# B&R Automation Studio project PT_KB_V01 (part 8)

### PGRad_Process.typ - not listed in the package file held
```iecst
TYPE
	E_RegulacijaBRB2 :
		( (* Regulaciona petlja pumpe koja doprema vodu iz BRB2. *) (* -------------------------------------------------------------------------- *) (* 1) Glavna stanja, izbor izvora i izbor aktivne opreme                     *)
		BRB2_00_NEAKTIVNA,
		BRB2_01_REG_PROTOK, (* Protok ka Podstanici/Hotelu. *)
		BRB2_02_REG_NIVO, (* Nivo prihvatnog suda. *)
		BRB2_03_REG_TEMPERATURA (* Temperatura sekundara izmenjivaca. *)
		);
	E_PGRad_State :
		( (* Glavna procesna stanja rada Podstanice prema izabranom izvoru. *)
		PG_00_Stand_By, (* Bez aktivnog izvora; izlazi su u bezbednom stanju i ceka se izbor/start. *)
		PG_01_Priprema_BRB2, (* Pokrece BRB2 i priprema ulaznu granu do potvrde pritiska/protoka. *)
		PG_02_Rad_BRB2, (* BRB2 napaja tank; aktivni su regulacija ulaza, izlazna pumpa i odzracivanje. *)
		PG_03_Zaustavljanje_BRB2, (* Kontrolisano ukida zahtev BRB2 i zatvara pripadajuce ventile. *)
		PG_11_Priprema_IEBKB1, (* Priprema IEBKB1 granu pre dozvole punjenja prihvatnog tanka. *)
		PG_12_Rad_IEBKB1, (* IEBKB1 je aktivni izvor i Podstanica vodi lokalnu regulaciju. *)
		PG_13_Zaustavljanje_IEBKB1, (* Kontrolisano zaustavlja IEBKB1 i zatvara njegovu ulaznu granu. *)
		PG_14_Transfer_IEBKB1_BRB2 (* Prebacuje napajanje sa IEBKB1 na prethodno pripremljeni BRB2. *)
		);
	E_BRB2PreparationState :
		( (* Stanja paralelne pripreme BRB2 pre transfera izvora. *)
		BRB2_PREP_00_IDLE, (* Priprema nije trazena; resetuju se privremene potvrde. *)
		BRB2_PREP_10_START, (* Poslat je start zahtev i ceka se potvrda protoka BRB2. *)
		BRB2_PREP_20_ZAGREVANJE, (* BRB2 ispira/zagreva cev do minimalne temperature. *)
		BRB2_PREP_30_SPReady, (* Protok i temperatura su potvrdeni; transfer izvora je dozvoljen. *)
		BRB2_PREP_40_STOPPING, (* Priprema se kontrolisano prekida i ceka se potvrda stopa. *)
		BRB2_PREP_90_FAULT (* Priprema je blokirana timeout-om ili procesnim interlockom. *)
		);
	E_RegulacionaVarijanta :
		( (* Izbor procesne velicine koju Podstanica regulise. *)
		_00_neaktivan, (* 0 - sve ugaseno, ni jedna varijanta nije izabrana. *)
		_01_REG_PRITISAK, (* 1 - PT vodi, prati zadati pritisak. *)
		_02_REG_NIVO (* 2 - PT vodi nivo prihvatnog tanka preko izlazne pumpe. *)
		);
	E_SelektovaniIzvor :
		( (* Izbor aktivnog izvora termalne vode za Podstanicu. *)
		_00_IZVOR_NIJE_IZABRAN, (* 0 - rezervisano za inicijalizaciju i dijagnostiku; binarni HMI selektor ne zadaje ovu vrednost. *)
		_01_BRB2, (* 1 - BRB2 kao izvor. *)
		_02_IEBKB1 (* 2 - IEBKB1 kao izvor. *)
		);
	E_AktivnaPumpaIzlazTanka :
		( (* Izbor aktivne izlazne pumpe prihvatnog tanka. *)
		_00_nijedna, (* 0 - nijedna pumpa aktivna na izlazu iz tanka. *)
		_01_Pu_PG_01, (* 1 - Pu_PG_01 aktivna. *)
		_02_Pu_PG_02 (* 2 - Pu_PG_02 aktivna. *)
		);
	E_AktivniPropVentilUlazTanka :
		( (* Izbor aktivnog proporcionalnog ventila na ulazu u tank. *) (* -------------------------------------------------------------------------- *) (* 2) Retentivni parametri procesa i pomocne runtime strukture                *)
		_00_PROP_VENTIL_NIJE_IZABRAN, (* 0 - nijedan prop. ventil nije izabran. *)
		_01_PG_PV01, (* 1 - PG_PV01 aktivan. *)
		_02_PG_PV02 (* 2 - PG_PV02 aktivan. *)
		);
	typCmdRetainUlazniVentiliPGRad : 	STRUCT  (* Zapamceni zahtevi bistabilnih ulaznih ventila PG_V01 i PG_V02. *)
		V01_Open : BOOL; (* PG_V01 - zapamceni zahtev IEBKB1 ulaznog ventila. *)
		V02_Open : BOOL; (* PG_V02 - zapamceni zahtev BRB2 ulaznog ventila. *)
	END_STRUCT;
	typParAirReleaseModePGRad : 	STRUCT  (* Parametri odzracivanja za jedan izvor vode. *)
		PV03 : typParAirRelease; (* Odzracivanje na ulazu termalne vode u podstanicu. *)
		PV04 : typParAirRelease; (* Odzracivanje na ulazu termalne vode u prihvatni tank. *)
	END_STRUCT;
	typParAirReleasePGRad : 	STRUCT  (* Grupisani parametri odzracivanja prema aktivnom izvoru. *)
		BRB2 : typParAirReleaseModePGRad; (* Parametri rada sa izvorom BRB2. *)
		IEBKB1 : typParAirReleaseModePGRad; (* Parametri rada sa izvorom IEBKB1. *)
	END_STRUCT;
	typTimeSPPGRad : 	STRUCT  (* Grupisani vremenski SP parametri u sekundama. *)
		PrelazPV05Cuvar_s : REAL; (* Vreme PT06 SP rampe [s]. *)
		OverlapPumpi_s : REAL; (* Maksimalno vreme paralelnog rada pri rotaciji [s]. *)
		AutoRestartDelay_s : REAL; (* Zadrzavanje pre automatskog starta [s]. *)
		ValvePositionTimeout_s : REAL; (* Maksimalno vreme hoda ventila [s]. *)
		InterlockDebounce_s : REAL; (* Vreme potvrde interlock povratnog signala [s]. *)
	END_STRUCT;
	typParBRB2PreparationPGRad : 	STRUCT  (* Paralelna priprema BRB2 dok IEBKB1 snabdeva tank. *)
		MinTemperature_degC : REAL; (* Minimalna temperatura TT_PG_07 za spremnost BRB2. *)
		MinFlow_lps : REAL; (* Minimalni potvrdeni protok BRB2 tokom zagrevanja. *)
		FlowTimeout_s : REAL; (* Maksimalno cekanje potvrde protoka nakon starta BRB2. *)
		TemperatureAlarm_s : REAL; (* Vreme do alarma ako temperatura nije dostignuta. *)
		TemperatureStopDelay_s : REAL; (* Dodatno vreme od alarma do kontrolisanog stopa. *)
		PressureAlarmDelay_s : REAL; (* Vreme visokog PT06 do alarma. *)
		PressureStopDelay_s : REAL; (* Dodatno vreme visokog PT06 do kontrolisanog stopa. *)
	END_STRUCT;
	typParTransferPGRad : 	STRUCT  (* Parametri transfera IEBKB1 na pripremljeni BRB2. *)
		PV05StartPressure_bar : REAL; (* Pocetni PT06 SP regulatora PG_PV05. *)
		PV05FinalPressure_bar : REAL; (* Krajnji PT06 SP regulatora PG_PV05. *)
		TankInletPressure_bar : REAL; (* Stalni PT04 SP aktivnog PG_PV01/PV02. *)
		PressureRamp_s : REAL; (* Trajanje rampe PT06 SP-a. *)
		FlowTimeout_s : REAL; (* Maksimalno cekanje potvrde BRB2 protoka pri transferu. *)
		PV05ClosedPercent : REAL; (* Otvorenost ispod koje se drenaÅ¾a smatra zatvorenom. *)
	END_STRUCT;
	typParPGRad : 	STRUCT  (* Zbirni procesni, vremenski i odzracni parametri Podstanice. *)
		SetPritisakPotisa : REAL; (* Zadati pritisak potisa glavne pumpe [bar]. *)
		MinProtok : REAL; (* Donja granica protoka. *)
		MaxProtok : REAL; (* Gornja granica protoka. *)
		MinFR_Pumpe : REAL; (* Minimalna frekvencija PID izlaza pumpi [Hz]. *)
		MaxFR_Pumpe : REAL; (* Maksimalna frekvencija PID izlaza pumpi [Hz]. *)
		SetPointNivoTanka : REAL; (* Ciljani nivo prihvatnog tanka [m]. *)
		SetPointNivoTankaUpozorenje : REAL; (* Informativni prag blizine fizickog preliva (~2.15-2.2m stvarnog preliva) [m]. *)
		SetPointMinTempIspiranja : REAL; (* Minimalna temperatura za zavrsetak ispiranja [degC]. *)
		SetPointPritisakPV05Ispiranje : REAL; (* PT06 SP tokom preispiranja [bar]. *)
		SetPointPritisakUlazTanka : REAL; (* PT04 SP aktivnog ulaznog ventila [bar]. *)
		SetPointMaxPritisakDolaznaCev : REAL; (* PT06 SP cuvara instalacije [bar]. *)
		PocetnaFrekvencaIzlaznePumpe : REAL; (* PID tracking frekvenca pri startu [Hz]. *)
		MaxOtvorPropZaZatvaranje : REAL; (* Najveca otvorenost za potvrdu zatvaranja [%]. *)
		BRB2Preparation : typParBRB2PreparationPGRad; (* Parametri nezavisnog zagrevanja BRB2. *)
		Transfer : typParTransferPGRad; (* Parametri kontrolisanog transfera izvora. *)
		TimeSP : typTimeSPPGRad; (* RETAIN vremenski SP parametri u sekundama. *)
		AirRelease : typParAirReleasePGRad; (* RETAIN parametri PV03/PV04 za oba izvora. *)
	END_STRUCT;
	typCtrlAirReleasePGRad : 	STRUCT  (* HMI i servisne komande jednog odzracnog ventila. *)
		EnableManual : BOOL; (* TRUE = direktna rucna komanda ima prioritet nad automatikom. *)
		ManualSP_Percent : REAL; (* Direktna rucna komanda ventila [%]. *)
		ResetAlarm : BOOL; (* Pojedinacni jednokratni reset memorisanog alarma. *)
	END_STRUCT;
	typAirReleaseChannelPGRad : 	STRUCT  (* Izvrsni FB i komande jednog odzracnog ventila. *)
		FB : FB_AirRelease; (* Instanca upravljanja odzracivanjem. *)
		Ctrl : typCtrlAirReleasePGRad; (* HMI i servisne komande instance. *)
	END_STRUCT;
	typAirReleasePGRad : 	STRUCT  (* Grupisane runtime instance odzracivanja PV03/PV04. *)
		PV03 : typAirReleaseChannelPGRad; (* Odzracivanje ulaza u podstanicu. *)
		PV04 : typAirReleaseChannelPGRad; (* Odzracivanje ulaza u prihvatni tank. *)
	END_STRUCT;
	typCtrlPGRad : 	STRUCT  (* Retentivni HMI izbori izvora, regulacije i aktivne opreme. *)
		SelektovaniIzvor : E_SelektovaniIzvor; (* Izbor izvora termalne vode. *)
		RegulacionaVarijanta : E_RegulacionaVarijanta; (* Izabrana regulaciona varijanta. *)
		AktivnaPumpaIzlazTanka : E_AktivnaPumpaIzlazTanka; (* Aktivna izlazna pumpa. *)
		AktivniPropVentilUlazTanka : E_AktivniPropVentilUlazTanka; (* Aktivni ulazni prop. ventil. *)
		AutoRestart : BOOL; (* Automatski start nakon cold boot-a. *)
		BRB2Regulacija : E_RegulacijaBRB2; (* Zaseban izbor regulacije pumpe BRB2; ne menja regulaciju izlaznih pumpi. *)
	END_STRUCT;
	typManualPGRad : 	STRUCT  (* Servisne rucne komande procesnih sekvenci Podstanice. *)
		Enable : BOOL; (* Dozvola servisnog rucnog rezima; aktivan samo u Standby. *)
		Sequence : USINT; (* Izabrana sekvenca: 1=BRB2 priprema/ispiranje, 2=IEBKB1 priprema, 3=kontrolisani stop. *)
		Start : BOOL; (* Impuls za pokretanje izabrane servisne sekvence. *)
		Stop : BOOL; (* Impuls za bezbedan prekid servisne sekvence. *)
		NextStep : BOOL; (* Impuls za zahtev sledeceg dozvoljenog podkoraka. *)
		Abort : BOOL; (* Impuls za povratak u Standby bez preskakanja stop logike. *)
	END_STRUCT;
END_TYPE

(* -------------------------------------------------------------------------- *)
(* 3) Krovni lokalni kontekst programa Rad_PG_KB                            *)
(* -------------------------------------------------------------------------- *)

TYPE
	typRadPGKBHmiCntrl : 	STRUCT  (* Komande automatskog rada iz HMI-ja Podstanice. *)
		Start : BOOL; (* Zahtev za pokretanje izabranog automatskog izvora. *)
		Stop : BOOL; (* Zahtev za kontrolisano zaustavljanje aktivnog izvora. *)
		Reset : BOOL; (* Zahtev za reset zakacenog procesnog fault-a. *)
		SelectIEBKB1 : BOOL; (* FALSE = BRB2 izvor; TRUE = IEBKB1 izvor. Prihvata se u Standby. *)
		SetDefaultParameters : BOOL; (* Jednokratni zahtev za vracanje RETAIN parametara na default vrednosti. *)
		PrepareBRB2 : BOOL; (* Zahtev za nezavisnu pripremu/zagrevanje BRB2 izvora. *)
		TransferToBRB2 : BOOL; (* Zahtev za transfer sa IEBKB1 na prethodno pripremljeni BRB2. *)
		Continue : BOOL; (* Zahtev za nastavak nakon potvrdenog protoka BRB2. *)
	END_STRUCT;
	typRadPGKBHmiManual : 	STRUCT  (* Komande servisnog manuelnog rada procesne sekvence. *)
		Enable : BOOL; (* Dozvola manuelnog rezima; koristi se samo kada je sekvenca u Standby. *)
		Sequence : USINT; (* Izbor manuelne sekvence: 1 = BRB2, 2 = IEBKB1. *)
		Start : BOOL; (* Impuls za pokretanje izabrane manuelne sekvence. *)
		Stop : BOOL; (* Impuls za kontrolisani prekid manuelne sekvence. *)
		NextStep : BOOL; (* Impuls za potvrdu sledeceg dozvoljenog podkoraka. *)
		Abort : BOOL; (* Impuls za prekid i povratak u bezbedni Standby. *)
	END_STRUCT;
	typRadPGKBHmi : 	STRUCT  (* Zbirni HMI interfejs lokalnog programa Rad_PG_KB. *)
		Cntrl : typRadPGKBHmiCntrl; (* Komande automatskog rada. *)
		Manual : typRadPGKBHmiManual; (* Komande servisnog manuelnog rada. *)
	END_STRUCT;
	typRadPGKBSequenceBRB2 : 	STRUCT  (* Lokalno stanje paralelne pripreme izvora BRB2. *)
		PreparationState : E_BRB2PreparationState; (* Stanje pripreme: start, zagrevanje, SP spreman, stop ili fault. *)
		PreparationSubstep : USINT; (* Aktivni podkorak pripreme BRB2. *)
		Ready : BOOL; (* TRUE kada su potvrdeni uslovi spremnosti BRB2 za transfer. *)
	END_STRUCT;
	typRadPGKBSequenceTransfer : 	STRUCT  (* Lokalna memorija zahteva transfera izvora. *)
		Requested : BOOL; (* Zakacen zahtev transfera do zavrsetka ili opoziva. *)
	END_STRUCT;
	typRadPGKBSequence : 	STRUCT  (* Izvrsni kontekst glavne state masine. *)
		State : E_PGRad_State; (* Aktivno glavno stanje rada Podstanice. *)
		Substep : USINT; (* Aktivni podkorak glavnog stanja; 0 je ulaz u stanje. *)
		BRB2 : typRadPGKBSequenceBRB2; (* Podstanje pripreme BRB2. *)
		Transfer : typRadPGKBSequenceTransfer; (* Podaci zahteva transfera IEBKB1 -> BRB2. *)
	END_STRUCT;
	typRadPGKBDiagFault : 	STRUCT  (* Zakacena procesna dijagnostika lokalne sekvence. *)
		Latched : BOOL; (* TRUE kada fault ostaje memorisan do dozvoljenog reset-a. *)
		Code : USINT; (* Numericki kod fault-a za HMI i komunikacioni status. *)
		Text : STRING[80]; (* Tekstualni opis aktivnog fault-a za operatera. *)
	END_STRUCT;
	typRadPGKBStatusPV05 : 	STRUCT  (* Status regulatora i funkcije PV05. *)
		FlushingOpened : BOOL; (* PT06 je dostigao uslov za dozvolu PV05 ispiranja. *)
	END_STRUCT;
	typRadPGKBStatusPump : 	STRUCT  (* Status izlazne pumpe prihvatnog tanka. *)
		OutletStopped : BOOL; (* Pumpa je u kontrolisanom praznjenju do donje granice histereze. *)
	END_STRUCT;
	typRadPGKBStatus : 	STRUCT  (* Izvedeni statusi lokalnih regulacionih funkcija. *)
		PV05 : typRadPGKBStatusPV05; (* Status PV05 funkcije. *)
		Pump : typRadPGKBStatusPump; (* Status izlazne pumpe. *)
		PrihvatniSudBlizuPreliva : BOOL; (* Informativno: nivo >= SetPointNivoTankaUpozorenje. Bez akcije/interlocka - ocekivano u pojedinim rezimima. *)
	END_STRUCT;
	typRadPGKBDiag : 	STRUCT  (* Zbirna dijagnostika programa Rad_PG_KB. *)
		Fault : typRadPGKBDiagFault; (* Zakaceni procesni fault. *)
	END_STRUCT;
	typRadPGKBControlPV05 : 	STRUCT  (* Izvrsna regulacija pritiska preko PV05. *)
		PID : MTBasicsPID; (* PID koji koristi PT06 kao PV i upravlja otvorenoscu PV05. *)
		FlushingSP : REAL; (* Trenutni rampirani SP pritiska PT06 [bar]. *)
	END_STRUCT;
	typRadPGKBControlPVUlazTanka : 	STRUCT  (* Izvrsna regulacija ulaznog proporcionalnog ventila. *)
		PID : MTBasicsPID; (* PID koji reguliše PT04 preko aktivnog PV01/PV02 ventila. *)
	END_STRUCT;
	typRadPGKBControl : 	STRUCT  (* Zbirni regulacioni FB-ovi programa Rad_PG_KB. *)
		PV05 : typRadPGKBControlPV05; (* Regulacija pritiska i cuvar PT06. *)
		PV_UlazTanka : typRadPGKBControlPVUlazTanka; (* Regulacija pritiska ulaza u prihvatni tank. *)
	END_STRUCT;
	typRadPGKBTimerValve : 	STRUCT  (* Tajmeri hoda PG_V01. *)
		Close : TON; (* Timeout potvrde zatvaranja PG_V01. *)
		Open : TON; (* Timeout potvrde otvaranja PG_V01. *)
	END_STRUCT;
	typRadPGKBTimerPGV02 : 	STRUCT  (* Tajmeri hoda PG_V02. *)
		Open : TON; (* Timeout potvrde otvaranja PG_V02. *)
		Close : TON; (* Timeout potvrde zatvaranja PG_V02. *)
	END_STRUCT;
	typRadPGKBTimerIEBKB1 : 	STRUCT  (* Tajmeri potvrde protoka izvora IEBKB1. *)
		StartProtokTimeout : TON; (* Maksimalno cekanje pocetka dotoka IEBKB1. *)
		ProtokNula : TON; (* Debounce potvrda da je protok IEBKB1 pao ispod praga. *)
		StopProtokTimeout : TON; (* Maksimalno cekanje prestanka dotoka IEBKB1. *)
	END_STRUCT;
	typRadPGKBTimerPGV05 : 	STRUCT  (* Tajmer zatvaranja izlaznog ventila PG_V05. *)
		Close : TON; (* Timeout potvrde zatvaranja PG_V05. *)
	END_STRUCT;
	typRadPGKBTimerBRB2 : 	STRUCT  (* Tajmeri nadzora pripreme izvora BRB2. *)
		PreparationFlow : TON; (* Timeout potvrde protoka BRB2 tokom pripreme. *)
		TemperatureAlarm : TON; (* Vreme do alarma ako temperatura BRB2 nije dostignuta. *)
		TemperatureStop : TON; (* Dodatno vreme do kontrolisanog stopa posle alarma temperature. *)
		PressureAlarm : TON; (* Vreme potvrde previsokog PT06 pritiska pre alarma. *)
		PressureStop : TON; (* Dodatno vreme do kontrolisanog stopa zbog PT06 pritiska. *)
	END_STRUCT;
	typRadPGKBTimerTransfer : 	STRUCT  (* Tajmeri kontrolisanog transfera izvora. *)
		PV05Guard : TON; (* Vreme rampe/cekanja promene PT06 SP-a. *)
		Flow : TON; (* Timeout potvrde BRB2 protoka tokom transfera. *)
	END_STRUCT;
	typRadPGKBTimer : 	STRUCT  (* Svi interni TON tajmeri programa Rad_PG_KB. *)
		PG_V01 : typRadPGKBTimerValve; (* Tajmeri ulaznog ventila IEBKB1. *)
		PG_V02 : typRadPGKBTimerPGV02; (* Tajmeri ulaznog ventila BRB2. *)
		PG_V05 : typRadPGKBTimerPGV05; (* Tajmer izlaznog/prelaznog ventila PG_V05. *)
		IEBKB1 : typRadPGKBTimerIEBKB1; (* Tajmeri protoka izvora IEBKB1. *)
		BRB2 : typRadPGKBTimerBRB2; (* Tajmeri pritiska, temperature i protoka BRB2. *)
		Transfer : typRadPGKBTimerTransfer; (* Tajmeri transfera i cuvara PT06. *)
	END_STRUCT;
	typRadPGKBAutoRestart : 	STRUCT  (* Automatski start nakon nestanka struje (WARMSTART), ako je PGRad.Ctrl.AutoRestart aktivan. *)
		WarmstartDetected : BOOL; (* Jednokratno zabelezeno u Init.st preko SysInfo.init_reason. *)
		Timer : TON; (* Odlozeni auto-start; PT = PGRad.Par.TimeSP.AutoRestartDelay_s. *)
	END_STRUCT;
	typRadPGKB : 	STRUCT  (* Krovni lokalni kontekst programa Rad_PG_KB. *)
		HMI : typRadPGKBHmi; (* HMI komande automatskog i manuelnog rada. *)
		Sequence : typRadPGKBSequence; (* Stanje glavne i pomocnih sekvenci. *)
		Control : typRadPGKBControl; (* Lokalni PID regulatori i njihove procesne vrednosti. *)
		Status : typRadPGKBStatus; (* Izvedeni statusi regulacije i aktuatora. *)
		Diag : typRadPGKBDiag; (* Fault status i tekst za HMI. *)
		Timer : typRadPGKBTimer; (* Interni tajmeri svih sekvenci. *)
		AutoRestart : typRadPGKBAutoRestart; (* Stanje automatskog starta posle WARMSTART-a. *)
	END_STRUCT;
END_TYPE

(* -------------------------------------------------------------------------- *)
(* 4) Procesne komande aktuatora i regulacioni ulazi                        *)
(* -------------------------------------------------------------------------- *)

TYPE
	typCmdOnOffPGRad : 	STRUCT  (* Procesni zahtevi otvaranja lokalnih ON/OFF ventila PG_V03..PG_V07. *)
		_03_Open : BOOL; (* PG_V03 - zahtev otvaranja izlazne grane pumpe 1. *)
		_04_Open : BOOL; (* PG_V04 - zahtev otvaranja izlazne grane pumpe 2. *)
		_05_Open : BOOL; (* PG_V05 - zahtev otvaranja bypass-a/preispiranja. *)
		_06_Open : BOOL; (* PG_V06 - zahtev otvaranja grane PV01 ka tanku. *)
		_07_Open : BOOL; (* PG_V07 - zahtev otvaranja grane PV02 ka tanku. *)
	END_STRUCT;
	typCmdPropVentilPGRad : 	STRUCT  (* Automatska dozvola i zahtev otvorenosti jednog proporcionalnog ventila. *)
		Enable : BOOL; (* Dozvola automatskog upravljanja ventilom. *)
		SP_Percent : REAL; (* Automatski zahtev otvorenosti 0..100%. *)
	END_STRUCT;
	typCmdPropVentiliPGRad : 	STRUCT  (* Grupisane procesne komande proporcionalnih ventila PG_PV01, PG_PV02 i PG_PV05. *)
		PV01 : typCmdPropVentilPGRad; (* PG_PV01 - ulazni proporcionalni ventil 1. *)
		PV02 : typCmdPropVentilPGRad; (* PG_PV02 - ulazni proporcionalni ventil 2. *)
		PV05 : typCmdPropVentilPGRad; (* PG_PV05 - drenazni proporcionalni ventil. *)
	END_STRUCT;
	typCmdAirReleaseChannelPGRad : 	STRUCT  (* Procesna dozvola jednog odzracnog ventila. *)
		Enable : BOOL; (* TRUE = dozvoljen automatski ili rucni rad FB_AirRelease. *)
	END_STRUCT;
	typCmdAirReleasePGRad : 	STRUCT  (* Komandni vektor odzracivanja iz state masine. *)
		PV03 : typCmdAirReleaseChannelPGRad; (* Dozvola odzracivanja ulaza u podstanicu. *)
		PV04 : typCmdAirReleaseChannelPGRad; (* Dozvola odzracivanja ulaza u tank. *)
		UseIEBKB1Parameters : BOOL; (* TRUE = koristi IEBKB1, FALSE = koristi BRB2 parametre. *)
		ResetAll : BOOL; (* Zajednicki reset oba FB-a iz KomandaReset. *)
	END_STRUCT;
	typCmdPumpaPGRad : 	STRUCT  (* Procesna dozvola rada jedne izlazne pumpe. *)
		Run : BOOL; (* Dozvola rada pumpe; frekvencu iskljucivo vodi PID_Pu_PT. *)
	END_STRUCT;
	typCmdPumpePGRad : 	STRUCT  (* Grupisane procesne komande izlaznih pumpi PG_Pu01 i PG_Pu02. *)
		_01 : typCmdPumpaPGRad; (* PG_Pu01 - komandni zahtev za izlaznu pumpu 1. *)
		_02 : typCmdPumpaPGRad; (* PG_Pu02 - komandni zahtev za izlaznu pumpu 2. *)
	END_STRUCT;
	typCmdPIDPumpePGRad : 	STRUCT  (* Ulazi i granice jedinog PID regulatora aktivne izlazne pumpe. *)
		Enable : BOOL; (* Dozvola rada PID_Pu_PT regulatora. *)
		ActValue : REAL; (* Aktivna regulisana vrednost: nivo tanka ili PT05 [m/bar]. *)
		SetValue : REAL; (* SP aktivne regulisane vrednosti [m/bar]. *)
		Invert : BOOL; (* Smer PID-a: TRUE za nivo, FALSE za pritisak. *)
		MaxOut : REAL; (* Maksimalni frekventni izlaz izabrane pumpe [Hz]. *)
		EnableTracking : BOOL; (* Dozvola bumpless starta na TrackingValue. *)
		TrackingValue : REAL; (* Pocetni frekventni zahtev PID-a pri startu [Hz]. *)
	END_STRUCT;
	typCmdPGRad : 	STRUCT  (* Neretentivni komandni vektor procesne state masine Podstanice. *)
		Aktivan : BOOL; (* State masina je vlasnik neretentivnih fizickih komandi. *)
		Ventili : typCmdOnOffPGRad; (* Zahtevi automatskih ON/OFF ventila. *)
		PropVentili : typCmdPropVentiliPGRad; (* Zahtevi proporcionalnih ventila. *)
		AirRelease : typCmdAirReleasePGRad; (* Zahtevi odzracivanja PV03/PV04. *)
		Pumpe : typCmdPumpePGRad; (* Zahtevi izlaznih pumpi. *)
		PID : typCmdPIDPumpePGRad; (* Ulazi jedinog PID-a izlazne pumpe. *)
	END_STRUCT;
END_TYPE

(* -------------------------------------------------------------------------- *)
(* 5) Statusni i retentivni kontekst Podstanice                              *)
(* -------------------------------------------------------------------------- *)

TYPE
	typPGRadStatus : 	STRUCT  (* Procesno stanje, podkorak i zakacena dijagnostika Podstanice. *)
		State : USINT; (* Eksplicitni PGRad state kod za komunikaciju i HMI. *)
		StateComment : STRING[80]; (* Operaterski opis aktivnog stanja. *)
		Substep : USINT; (* Aktivni podkorak state masine. *)
		SubstepComment : STRING[80]; (* Operaterski opis aktivnog podkoraka. *)
		Fault : BOOL; (* Zakacena procesna greska. *)
		FaultCode : USINT; (* Sifra zakacene procesne greske. *)
		BRB2PreparationState : USINT; (* Nezavisno stanje pripreme BRB2. *)
		BRB2PreparationStateComment : STRING[80]; (* Tekstualni opis nezavisnog stanja pripreme BRB2. *)
		BRB2Ready : BOOL; (* Temperatura, protok i minimalno trajanje su potvrdeni. *)
		IEBKB1InterfaceReady : BOOL; (* Buduci IEBKB1 ugovor je kompletan i validan. *)
		TransferBlocked : BOOL; (* Transfer je blokiran zbog nepotpunog IEBKB1 ugovora ili interlocka. *)
	END_STRUCT;
	typPGRad : 	STRUCT  (* Retentivni kontekst komandi, parametara i HMI izbora Podstanice. *)
		CmdRetain : typCmdRetainUlazniVentiliPGRad; (* Retain komande bistabilnih ulaznih ventila. *)
		Par : typParPGRad; (* Retain projektni parametri procesa podstanice. *)
		Ctrl : typCtrlPGRad; (* Retain HMI izbor izvora i regulacije. *)
	END_STRUCT;
END_TYPE
```

### Alarm.var - not listed in the package file held
```iecst
VAR
	PT_Alarm : typPTAlarm; (* Centralni alarmni status i komande Podstanice. *)
END_VAR
```

### PG_IO.var - not listed in the package file held
```iecst
VAR
	PG : PG_type; (* Korenski I/O i HMI objekat podstanice. *)
END_VAR
```

### PGRad_Communication.var - not listed in the package file held
```iecst
VAR
	PGRad_BRB2Cmd : typVezaPGRadBRB2; (* Kanonski PT izlazni status. *)
	PGRad_BRB2 : typVezaPGRadBRB2; (* Lokalni procesni komunikacioni ugovor. *)
	PGRad_BRB2_Tx : typVezaPGRadBRB2; (* PT izlazni AsIMA snapshot. *)
	PGRad_BRB2_Rx : typVezaPGRadBRB2; (* BRB2 ulazni AsIMA snapshot. *)
	PGRad_BRB2Watchdog : typBRB2CommWatchdog; (* Nadzor BRB2 StatusCounter-a. *)
	PGRad_IEBKB1Prepared : typIEBKB1PreparedInterface; (* Buduci IEBKB1 ugovor. *)
END_VAR
```

### PGRad_HMI.var - not listed in the package file held
```iecst
VAR
	PGRad_Status : typPGRadStatus; (* Procesni status za HMI. *)
	PGRad_TrendCursor : typPGRadTrendCursor; (* HMI trend kursor. *)
END_VAR
```

### PGRad_Process.var - not listed in the package file held
```iecst
VAR RETAIN
	PGRad : typPGRad; (* Retain procesni kontekst: Ctrl, Par i CmdRetain. *)
END_VAR

VAR
	AktivniUlazniProtok : REAL; (* Realni protok aktivnog izvora termalne vode [l/s]. *)
	Predata_Snaga : REAL; (* Ukupna snaga predata izmenjivacima [kW]. *)
	Snaga_grejanja_hotela : REAL; (* Snaga predata hotelskom grejanju [kW]. *)
	Snaga_sanitarnog_grejanja : REAL; (* Preostala snaga predata sanitarnom grejanju [kW]. *)
	DP_Izmejnivac : REAL; (* DeviceCtrl racuna diferencijalni pritisak velikog izmenjivaca [bar]. *)
	DP_strainer : REAL; (* DeviceCtrl racuna diferencijalni pritisak grubog filtera [bar]. *)
	NivoPrihvatniSud : REAL; (* DeviceCtrl racuna hidrostaticki nivo prihvatnog suda [m]. *)
	PID_Pu_PT : MTBasicsPID; (* PID petlja pumpi na izlazu iz prihvatnog tanka. *)
	PGRad_Cmd : typCmdPGRad; (* Neretentivni komandni vektor state masine. *)
	PGRad_AirRelease : typAirReleasePGRad; (* Runtime odzracivanje PV03/PV04. *)
END_VAR
```

### Program Logical/CAN (IEC)

#### Cyclic.st - Cyclic code
```iecst
PROGRAM _CYCLIC
	(* ======================================================================== *)
	(* CAN - UPRAVLJANJE PG_PU01 I PG_PU02                                  *)
	(* COMMON: prenosi granice, nazivnu snagu i reset komandu ka CAN FB-u.    *)
	(* AUTO/MANUAL: CAN sloj ne bira rezim; koristi vec formirani Start/FR_set. *)
	(* STOP/FAULT: CAN alarmi se vracaju u status pumpe i alarmni sloj.        *)
	(* STATUS: Running, brzina, snaga, struja i alarmi se objavljuju lokalno.  *)
	(* ======================================================================== *)
	(* -------------------------------------------------------------------------- *)
	(* 1) PG_Pu01 CANopen upravljanje                                              *)
	(* -------------------------------------------------------------------------- *)
	PG.Act.Pu._1.CAN_FB.b_Enable := PG.Act.Pu._1.Enable;
	PG.Act.Pu._1.CAN_FB.b_Start := PG.Act.Pu._1.Start;
	PG.Act.Pu._1.CAN_FB.b_AlarmRst := PG.Act.Pu._1.Reset_Alarm OR PT_Alarm.ResetPulse.Devices;
	PG.Act.Pu._1.CAN_FB.w_FR_min := PG.Act.Pu._1.FR_min;
	PG.Act.Pu._1.CAN_FB.w_FR_max := PG.Act.Pu._1.FR_max;
	PG.Act.Pu._1.CAN_FB.w_NomSnaga := PG.Act.Pu._1.Motor_Nominalna_Snaga;
	PG.Act.Pu._1.CAN_FB.w_ZadataBrzHz := PG.Act.Pu._1.FR_set;
	PG.Act.Pu._1.CAN_FB();
	PG.Act.Pu._1.Status_inRun := PG.Act.Pu._1.CAN_FB.b_Running;
	PG.Act.Pu._1.Alarm_FR := PG.Act.Pu._1.CAN_FB.b_Alarm_FR;
	PG.Act.Pu._1.Alarm_CAN := PG.Act.Pu._1.CAN_FB.b_Alarm_CAN;
	PG.Act.Pu._1.Ostvarena_brzina := PG.Act.Pu._1.CAN_FB.w_MotorBrz;
	PG.Act.Pu._1.Motor_Snaga := PG.Act.Pu._1.CAN_FB.w_MotorSnaga;
	PG.Act.Pu._1.Motor_Struja := PG.Act.Pu._1.CAN_FB.w_MotorStruja;

	(* -------------------------------------------------------------------------- *)
	(* 2) PG_Pu02 CANopen upravljanje                                              *)
	(* -------------------------------------------------------------------------- *)
	PG.Act.Pu._2.CAN_FB.b_Enable := PG.Act.Pu._2.Enable;
	PG.Act.Pu._2.CAN_FB.b_Start := PG.Act.Pu._2.Start;
	PG.Act.Pu._2.CAN_FB.b_AlarmRst := PG.Act.Pu._2.Reset_Alarm OR PT_Alarm.ResetPulse.Devices;
	PG.Act.Pu._2.CAN_FB.w_FR_min := PG.Act.Pu._2.FR_min;
	PG.Act.Pu._2.CAN_FB.w_FR_max := PG.Act.Pu._2.FR_max;
	PG.Act.Pu._2.CAN_FB.w_NomSnaga := PG.Act.Pu._2.Motor_Nominalna_Snaga;
	PG.Act.Pu._2.CAN_FB.w_ZadataBrzHz := PG.Act.Pu._2.FR_set;
	PG.Act.Pu._2.CAN_FB();
	PG.Act.Pu._2.Status_inRun := PG.Act.Pu._2.CAN_FB.b_Running;
	PG.Act.Pu._2.Alarm_FR := PG.Act.Pu._2.CAN_FB.b_Alarm_FR;
	PG.Act.Pu._2.Alarm_CAN := PG.Act.Pu._2.CAN_FB.b_Alarm_CAN;
	PG.Act.Pu._2.Ostvarena_brzina := PG.Act.Pu._2.CAN_FB.w_MotorBrz;
	PG.Act.Pu._2.Motor_Snaga := PG.Act.Pu._2.CAN_FB.w_MotorSnaga;
	PG.Act.Pu._2.Motor_Struja := PG.Act.Pu._2.CAN_FB.w_MotorStruja;
END_PROGRAM
```

### Program Logical/Config2_ATV (IEC)

#### Init.st - Init code
```iecst
PROGRAM _INIT
	(* -------------------------------------------------------------------------- *)
	(* 1) Config2 CANopen parametri izlaznih pumpi                                *)
	(* -------------------------------------------------------------------------- *)
	PG.Act.Pu._1.Enable := TRUE;
	PG.Act.Pu._1.FR_min := 10.0; (* Minimalna dozvoljena frekvencija PG_Pu01 [Hz]. *)
	PG.Act.Pu._1.FR_max := 50.0; (* Maksimalna dozvoljena frekvencija PG_Pu01 [Hz]. *)
	PG.Act.Pu._1.Motor_Nominalna_Snaga := 7.5; (* Nazivna snaga motora PG_Pu01 [kW]. *)

	PG.Act.Pu._2.Enable := TRUE;
	PG.Act.Pu._2.FR_min := 10.0; (* Minimalna dozvoljena frekvencija PG_Pu02 [Hz]. *)
	PG.Act.Pu._2.FR_max := 50.0; (* Maksimalna dozvoljena frekvencija PG_Pu02 [Hz]. *)
	PG.Act.Pu._2.Motor_Nominalna_Snaga := 7.5; (* Nazivna snaga motora PG_Pu02 [kW]. *)
END_PROGRAM
```

### Program Logical/PID_Pu_PT

#### Cyclic.st
```iecst
PROGRAM _CYCLIC
	(* ======================================================================== *)
	(* PID_Pu_PT_CYCLIC                                                           *)
	(* PID petlja pumpi na izlazu iz prihvatnog tanka.                            *)
	(* ======================================================================== *)

	(* -------------------------------------------------------------------------- *)
	(* 1) Rad po komandi state masine: PID je jedini vlasnik frekvencije i Run-a. *)
	(* -------------------------------------------------------------------------- *)
	(* Donja granica PID izlaza centralno se preuzima iz parametara pumpi. *)
	PID_Pu_PT.MinOut := PGRad.Par.MinFR_Pumpe;

	IF PGRad_Cmd.Aktivan THEN
		(* 1.1) Prenos procesnog zahteva u PID regulator. *)
		PID_Pu_PT.Enable := PGRad_Cmd.PID.Enable;
		PID_Pu_PT.ActValue := PGRad_Cmd.PID.ActValue;
		PID_Pu_PT.SetValue := PGRad_Cmd.PID.SetValue;
		PID_Pu_PT.Invert := PGRad_Cmd.PID.Invert;
		PID_Pu_PT.MaxOut := PGRad_Cmd.PID.MaxOut; (* Preuzima PGRad.Par.MaxFR_Pumpe. *)
		PID_Pu_PT.EnableTracking := PGRad_Cmd.PID.EnableTracking;
		PID_Pu_PT.TrackingValue := PGRad_Cmd.PID.TrackingValue;
		IF EDGEPOS(PGRad_Cmd.PID.Enable) THEN
			PID_Pu_PT.Update := TRUE;
		END_IF
		PID_Pu_PT();
		IF PID_Pu_PT.UpdateDone THEN
			PID_Pu_PT.Update := FALSE;
		END_IF

		(* 1.2) Iskljucivo izabrana izlazna pumpa dobija PID frekvenciju i Run. *)
		PG.Act.Pu._1.Start := FALSE;
		PG.Act.Pu._2.Start := FALSE;
		IF PGRad_Cmd.PID.Enable THEN
			IF PGRad_Cmd.Pumpe._01.Run THEN
				PG.Act.Pu._1.FR_set := PID_Pu_PT.Out;
				PG.Act.Pu._1.Start := TRUE;
			ELSIF PGRad_Cmd.Pumpe._02.Run THEN
				PG.Act.Pu._2.FR_set := PID_Pu_PT.Out;
				PG.Act.Pu._2.Start := TRUE;
			END_IF
		END_IF

	ELSE
		(* -------------------------------------------------------------------------- *)
		(* 2) Rucni rad pumpi                                                       *)
		(* -------------------------------------------------------------------------- *)
		(* U rucnom rezimu HMI neposredno zadaje Start i FR_set izabrane pumpe. *)
		PID_Pu_PT.Enable := FALSE;
		PID_Pu_PT.EnableTracking := FALSE;
		PID_Pu_PT();

		(* -------------------------------------------------------------------------- *)
		(* 3) Zadrzavanje postojeceg nasledjenog bypass zahteva                     *)
		(* -------------------------------------------------------------------------- *)
		(* PG_V05 prati otvoren ulazni ventil PG_V01 u nasledjenom lokalnom rezimu. *)
		IF PG.Act.AV._1.Open THEN
			PG.Act.AV._5.Open := TRUE;
		END_IF
	END_IF
END_PROGRAM
```

#### Exit.st
```iecst
PROGRAM _EXIT
	(* ======================================================================== *)
	(* PID_Pu_PT_EXIT                                                             *)
	(* PID petlja pumpi na izlazu iz prihvatnog tanka.                            *)
	(* Nema posebne EXIT akcije; Run i frekvencu vlasnicki postavlja CYCLIC.     *)
	(* ======================================================================== *)

END_PROGRAM
```

### Program Logical/Project/IO (IEC)

#### Cyclic.st
```iecst
PROGRAM _CYCLIC

(* ============================================================================ *)
(* IO_CYCLIC  Pozivi svih BR_Lib FB instanci                                   *)
(* Objekat: PG  Podstanica grejanja 1, Kursumlijska Banja                     *)
(* Sva IO mapiranja su u IoMap.iom  ovde su samo pozivi FB-ova.               *)
(* Redosled: senzori -> DI -> AV -> RV -> PV -> Pu                            *)
(* ============================================================================ *)

(* -------------------------------------------------------------------------- *)
(* 1) FBAI01_DI01  Senzori pritiska Pt (_0_0, _1.._6, _NS1, _NS2)            *)
(* Skaliranje raw AI -> bar. Parametri postavljeni u IO_Init.                 *)
(* -------------------------------------------------------------------------- *)
PG.Sens.Pt._0_0();  (* Pritisak komprimovanog vazduha, skalirani opseg -1 do 14 [bar] *)
PG.Sens.Pt._1();    (* Pritisak termalne vode na ulazu u podstanicu [bar] *)
PG.Sens.Pt._2();    (* Pritisak termalne vode posle streinera grubih filtera [bar] *)
PG.Sens.Pt._3();    (* Pritisak termalne vode posle velikog izmenjivaca [bar] *)
PG.Sens.Pt._4();    (* Pritisak termalne vode na ulazu u prihvatni tank [bar] *)
PG.Sens.Pt._5();    (* Pritisak na potisu transportnih pumpi [bar] *)
PG.Sens.Pt._6();    (* Dodatni transmiter pritiska [bar] *)
PG.Sens.Pt._NS1();  (* Pritisak na dnu prihvatnog tanka [bar] *)
PG.Sens.Pt._NS2();  (* Pritisak na vrhu prihvatnog tanka [bar] *)

(* -------------------------------------------------------------------------- *)
(* 2) FBAI01_DI01  Temperature TT_PG_01..TT_PG_11                         *)
(* Svi kanali su fizicki mapirani na X20AI4622b, X67AI1323 i X67AI1333b.    *)
(* -------------------------------------------------------------------------- *)
PG.Sens.Tt._1();  (* TT_PG_01 - ulaz u veliki razmenjivac PGRT01 [degC]. *)
PG.Sens.Tt._2();  (* TT_PG_02 - ulaz u prihvatni tank [degC]. *)
PG.Sens.Tt._3();  (* TT_PG_03 - temperatura u prihvatnom tanku [degC]. *)
PG.Sens.Tt._4();  (* TT_PG_04 - izlaz iz velikog razmenjivaca PGRT01 [degC]. *)
PG.Sens.Tt._5();  (* TT_PG_05 - ulaz u mali razmenjivac PGRT02 [degC]. *)
PG.Sens.Tt._6();  (* TT_PG_06 - izlaz iz malog razmenjivaca PGRT02 [degC]. *)
PG.Sens.Tt._7();  (* TT_PG_07 - drenazni vod za potvrdu zavrsetka preispiranja [degC]. *)
PG.Sens.Tt._8();  (* TT_PG_08 - ulaz tehnicke vode u direktni izmenjivac [degC]. *)
PG.Sens.Tt._9();  (* TT_PG_09 - izlaz tehnicke vode iz direktnog izmenjivaca [degC]. *)
PG.Sens.Tt._10(); (* TT_PG_10 - ulaz sanitarne vode u direktni izmenjivac [degC]. *)
PG.Sens.Tt._11(); (* TT_PG_11 - izlaz sanitarne vode iz direktnog izmenjivaca [degC]. *)

(* -------------------------------------------------------------------------- *)
(* 3) FBAI01_DI01  Merac protoka MP (_1)                                      *)
(* Skaliranje raw AI -> m3/h. TransmitterStatus DI aktivan (EnableStatusCheck).*)
(* -------------------------------------------------------------------------- *)
PG.Sens.MP._1();  (* Merac protoka na potisu tople termalne vode ka potrosacima [m3/h] *)

(* -------------------------------------------------------------------------- *)
(* 4) FB_DI  Nivo prekidaci LS (_1.._5)                                       *)
(* DI detekcija prisustva tecnosti u odzraci. DelayOn/Off=T#1s.               *)
(* -------------------------------------------------------------------------- *)
PG.Sens.LS._1();  (* Nizak nivo vode u prihvatnom tanku za rad pumpi *)
PG.Sens.LS._2();  (* Donji nivo u odzracnom cilindru na ulazu vode u podstanicu *)
PG.Sens.LS._3();  (* Gornji nivo u odzracnom cilindru na ulazu vode u podstanicu *)
PG.Sens.LS._4();  (* Donji nivo u odzracnom cilindru na ulazu vode u prihvatni tank *)
PG.Sens.LS._5();  (* Gornji nivo u odzracnom cilindru na ulazu vode u prihvatni tank *)

(* -------------------------------------------------------------------------- *)
(* 5) FB_DI  Prestrujni ventili OWF (_1, _2)                                  *)
(* DI povratni signal otvorenog polozaja. DelayOn/Off=T#500ms.                *)
(* -------------------------------------------------------------------------- *)
PG.Sens.OWF._1();  (* Zastitni prestrujni ventil od hidraulickog udara 1 *)
PG.Sens.OWF._2();  (* Zastitni prestrujni ventil od hidraulickog udara 2 *)

(* -------------------------------------------------------------------------- *)
(* 6) FB_V_EMV + FB_V_ON_OFF_FB  Automatski ventili AV (_1.._7)               *)
(* AV._1/2: bistabilni - CmdOpen i CmdClose mapirani u IoMap.                 *)
(* AV._3..AV._7: spring-return NC - samo Cmd mapiran u IoMap.                 *)
(* -------------------------------------------------------------------------- *)
PG.Act.AV._1();  (* Elektromotorni bistabilni leptir ventil DN125, OpenMaxTime=20s *)
PG.Act.AV._2();  (* Elektromotorni bistabilni leptir ventil DN125, OpenMaxTime=20s *)
PG.Act.AV._3();  (* Pneumatski NC spring-return leptir ventil DN125, OpenMaxTime=10s *)
PG.Act.AV._4();  (* Pneumatski NC spring-return leptir ventil DN125, OpenMaxTime=10s *)
PG.Act.AV._5();  (* Pneumatski NC spring-return leptir ventil DN125, OpenMaxTime=10s *)
PG.Act.AV._6();  (* Pneumatski NC spring-return leptir ventil DN125, OpenMaxTime=10s *)
PG.Act.AV._7();  (* Pneumatski NC spring-return leptir ventil DN125, OpenMaxTime=10s *)

(* -------------------------------------------------------------------------- *)
(* 7) FB_HV_2LS  Rucni leptir ventili RV (_19, _21.._27)                     *)
(* Monitoring 2 krajnja prekidaca, alarm pri timeout tranziciji.              *)
(* -------------------------------------------------------------------------- *)
PG.Act.RV._19();  (* Rucni ventil posle membranskog ventila PG_PV01 *)
PG.Act.RV._21();  (* Rucni ventil posle membranskog ventila PG_PV02 *)
PG.Act.RV._22();  (* Drenazni total ventil na dnu prihvatnog tanka *)
PG.Act.RV._23();  (* Ulaz u Pumpu PG_Pu01 *)
PG.Act.RV._24();  (* Ulaz u Pumpu PG_Pu02 *)
PG.Act.RV._25();  (* Bajpasni izlaz iz tanka ka instalaciji za izbacivanje gasa van kotlarnice *)
PG.Act.RV._26();  (* Ulaz u vakuum pumpu *)
PG.Act.RV._27();  (* Izlaz iz vakuum pumpe ka instalaciji za izbacivanje gasa van kotlarnice *)

(* -------------------------------------------------------------------------- *)
(* 8) FB_PvAiAo_Fast  Proporcionalni membranski ventili PV (_1.._5)           *)
(* AI_Raw povratni signal i AO_Raw komanda direktno mapirani u IoMap.         *)
(* -------------------------------------------------------------------------- *)

	PG.Act.PV._1(); (* Obrada granica, izbora Manual/Auto i AO komande PV._1. *)

	PG.Act.PV._2(); (* Obrada granica, izbora Manual/Auto i AO komande PV._2. *)

	PG.Act.PV._3(); (* Obrada granica, izbora Manual/Auto i AO komande PV._3. *)

	PG.Act.PV._4(); (* Obrada granica, izbora Manual/Auto i AO komande PV._4. *)

	PG.Act.PV._5(); (* Obrada granica, izbora Manual/Auto i AO komande PV._5. *)

END_PROGRAM
```

#### Init.st
```iecst
PROGRAM _INIT

(* ============================================================================ *)
(* IO_INIT  Inicijalizacija parametara za sve BR_Lib FB instance               *)
(* Objekat: PG  Podstanica grejanja 1, Kursumlijska Banja                     *)
(* IO veze: IoMap.iom  ovde su samo parametri i Enable politika.              *)
(* ============================================================================ *)

(* -------------------------------------------------------------------------- *)
(* 1) FBAI01_DI01  Senzori pritiska Pt (_1.._6)                               *)
(* X20AI4622 / X20AI4622a, 4-20mA, Cerabar PMP23. Opseg: -1...9 bara.        *)
(* ScaledMin=-1.0: zastitni offset jer 4mA odgovara 0 bara na terenu.        *)
(* -------------------------------------------------------------------------- *)
(* Pt._0_0: Pritisak komprimovanog vazduha [bar] *)
PG.Sens.Pt._0_0.AI_Input.Enable             := TRUE;      (* aktivira FB, pokrece skaliranje i statusnu logiku *)
PG.Sens.Pt._0_0.AI_Param.RawMin             := 0;         (* donja granica raw ADC opsega (0 = 4mA) *)
PG.Sens.Pt._0_0.AI_Param.RawMax             := 32767;     (* gornja granica raw ADC opsega (32767 = 20mA) *)
PG.Sens.Pt._0_0.AI_Param.ScaledMin          := -1.0;      (* donja fizicka vrednost opsega [bar] *)
PG.Sens.Pt._0_0.AI_Param.ScaledMax          := 15.0;      (* gornja fizicka vrednost opsega [bar] *)
PG.Sens.Pt._0_0.AI_Param.UnitOfMeasure      := 'bar';     (* jedinica za prikaz na HMI *)
PG.Sens.Pt._0_0.AI_Param.EnableStatusCheck  := FALSE;     (* bez TransmitterStatus DI - nije prikljucen *)

(* Pt._1: Pritisak termalne vode na ulazu u podstanicu [bar] *)
PG.Sens.Pt._1.AI_Input.Enable             := TRUE;      (* aktivira FB, pokrece skaliranje i statusnu logiku *)
PG.Sens.Pt._1.AI_Param.RawMin             := 0;         (* donja granica raw ADC opsega (0 = 4mA) *)
PG.Sens.Pt._1.AI_Param.RawMax             := 32767;     (* gornja granica raw ADC opsega (32767 = 20mA) *)
PG.Sens.Pt._1.AI_Param.ScaledMin          := -1.0;      (* 0-10 bar, offset -1: 4mA = 0 bar na terenu *)
PG.Sens.Pt._1.AI_Param.ScaledMax          := 9.0;       (* gornja fizicka vrednost opsega [bar] *)
PG.Sens.Pt._1.AI_Param.UnitOfMeasure      := 'bar';     (* jedinica za prikaz na HMI *)
PG.Sens.Pt._1.AI_Param.EnableStatusCheck  := FALSE;     (* bez TransmitterStatus DI - nije prikljucen *)

(* Pt._2: Pritisak termalne vode posle streinera grubih filtera [bar] *)
PG.Sens.Pt._2.AI_Input.Enable             := TRUE;      (* aktivira FB, pokrece skaliranje i statusnu logiku *)
PG.Sens.Pt._2.AI_Param.RawMin             := 0;         (* donja granica raw ADC opsega (0 = 4mA) *)
PG.Sens.Pt._2.AI_Param.RawMax             := 32767;     (* gornja granica raw ADC opsega (32767 = 20mA) *)
PG.Sens.Pt._2.AI_Param.ScaledMin          := -1.0;      (* 0-10 bar, offset -1: 4mA = 0 bar na terenu *)
PG.Sens.Pt._2.AI_Param.ScaledMax          := 9.0;       (* gornja fizicka vrednost opsega [bar] *)
PG.Sens.Pt._2.AI_Param.UnitOfMeasure      := 'bar';     (* jedinica za prikaz na HMI *)
PG.Sens.Pt._2.AI_Param.EnableStatusCheck  := FALSE;     (* bez TransmitterStatus DI - nije prikljucen *)

(* Pt._3: Pritisak termalne vode posle velikog izmenjivaca [bar] *)
PG.Sens.Pt._3.AI_Input.Enable             := TRUE;      (* aktivira FB, pokrece skaliranje i statusnu logiku *)
PG.Sens.Pt._3.AI_Param.RawMin             := 0;         (* donja granica raw ADC opsega (0 = 4mA) *)
PG.Sens.Pt._3.AI_Param.RawMax             := 32767;     (* gornja granica raw ADC opsega (32767 = 20mA) *)
PG.Sens.Pt._3.AI_Param.ScaledMin          := -1.0;      (* 0-10 bar, offset -1: 4mA = 0 bar na terenu *)
PG.Sens.Pt._3.AI_Param.ScaledMax          := 9.0;       (* gornja fizicka vrednost opsega [bar] *)
PG.Sens.Pt._3.AI_Param.UnitOfMeasure      := 'bar';     (* jedinica za prikaz na HMI *)
PG.Sens.Pt._3.AI_Param.EnableStatusCheck  := FALSE;     (* bez TransmitterStatus DI - nije prikljucen *)

(* Pt._4: Pritisak termalne vode na ulazu u prihvatni tank [bar] *)
PG.Sens.Pt._4.AI_Input.Enable             := TRUE;      (* aktivira FB, pokrece skaliranje i statusnu logiku *)
PG.Sens.Pt._4.AI_Param.RawMin             := 0;         (* donja granica raw ADC opsega (0 = 4mA) *)
PG.Sens.Pt._4.AI_Param.RawMax             := 32767;     (* gornja granica raw ADC opsega (32767 = 20mA) *)
PG.Sens.Pt._4.AI_Param.ScaledMin          := -1.0;      (* 0-10 bar, offset -1: 4mA = 0 bar na terenu *)
PG.Sens.Pt._4.AI_Param.ScaledMax          := 9.0;       (* gornja fizicka vrednost opsega [bar] *)
PG.Sens.Pt._4.AI_Param.UnitOfMeasure      := 'bar';     (* jedinica za prikaz na HMI *)
PG.Sens.Pt._4.AI_Param.EnableStatusCheck  := FALSE;     (* bez TransmitterStatus DI - nije prikljucen *)

(* Pt._5: Pritisak na potisu transportnih pumpi [bar] *)
PG.Sens.Pt._5.AI_Input.Enable             := TRUE;      (* aktivira FB, pokrece skaliranje i statusnu logiku *)
PG.Sens.Pt._5.AI_Param.RawMin             := 0;         (* donja granica raw ADC opsega (0 = 4mA) *)
PG.Sens.Pt._5.AI_Param.RawMax             := 32767;     (* gornja granica raw ADC opsega (32767 = 20mA) *)
PG.Sens.Pt._5.AI_Param.ScaledMin          := -1.0;      (* 0-10 bar, offset -1: 4mA = 0 bar na terenu *)
PG.Sens.Pt._5.AI_Param.ScaledMax          := 9.0;       (* gornja fizicka vrednost opsega [bar] *)
PG.Sens.Pt._5.AI_Param.UnitOfMeasure      := 'bar';     (* jedinica za prikaz na HMI *)
PG.Sens.Pt._5.AI_Param.EnableStatusCheck  := FALSE;     (* bez TransmitterStatus DI - nije prikljucen *)

(* Pt._6: Dodatni transmiter pritiska [bar] *)
PG.Sens.Pt._6.AI_Input.Enable             := TRUE;      (* aktivira FB, pokrece skaliranje i statusnu logiku *)
PG.Sens.Pt._6.AI_Param.RawMin             := 0;         (* donja granica raw ADC opsega (0 = 4mA) *)
PG.Sens.Pt._6.AI_Param.RawMax             := 32767;     (* gornja granica raw ADC opsega (32767 = 20mA) *)
PG.Sens.Pt._6.AI_Param.ScaledMin          := -1.0;      (* 0-10 bar, offset -1: 4mA = 0 bar na terenu *)
PG.Sens.Pt._6.AI_Param.ScaledMax          := 9.0;       (* gornja fizicka vrednost opsega [bar] *)
PG.Sens.Pt._6.AI_Param.UnitOfMeasure      := 'bar';     (* jedinica za prikaz na HMI *)
PG.Sens.Pt._6.AI_Param.EnableStatusCheck  := FALSE;     (* bez TransmitterStatus DI - nije prikljucen *)

(* -------------------------------------------------------------------------- *)
(* 2) FBAI01_DI01  Senzori niskog pritiska Pt (_NS1, _NS2) za merenje nivoa  *)
(* X20AI4622a, 4-20mA, Cerabar PMP23. Opseg: -0.1...0.3 bar (PTNS).          *)
(* -------------------------------------------------------------------------- *)
(* Pt._NS1: Pritisak na dnu prihvatnog tanka [bar] *)
PG.Sens.Pt._NS1.AI_Input.Enable             := TRUE;    (* aktivira FB, pokrece skaliranje i statusnu logiku *)
PG.Sens.Pt._NS1.AI_Param.RawMin             := 0;       (* donja granica raw ADC opsega (0 = 4mA) *)
PG.Sens.Pt._NS1.AI_Param.RawMax             := 32767;   (* gornja granica raw ADC opsega (32767 = 20mA) *)
PG.Sens.Pt._NS1.AI_Param.ScaledMin          := -0.1;  (* donja fizicka vrednost opsega [bar] *)
PG.Sens.Pt._NS1.AI_Param.ScaledMax          := 0.3;   (* gornja fizicka vrednost opsega [bar] *)
PG.Sens.Pt._NS1.AI_Param.UnitOfMeasure      := 'bar';  (* jedinica za prikaz na HMI *)
PG.Sens.Pt._NS1.AI_Param.EnableStatusCheck  := FALSE;   (* bez TransmitterStatus DI - nije prikljucen *)

(* Pt._NS2: Pritisak na vrhu prihvatnog tanka [bar] *)
PG.Sens.Pt._NS2.AI_Input.Enable             := TRUE;    (* aktivira FB, pokrece skaliranje i statusnu logiku *)
PG.Sens.Pt._NS2.AI_Param.RawMin             := 0;       (* donja granica raw ADC opsega (0 = 4mA) *)
PG.Sens.Pt._NS2.AI_Param.RawMax             := 32767;   (* gornja granica raw ADC opsega (32767 = 20mA) *)
PG.Sens.Pt._NS2.AI_Param.ScaledMin          := -0.1;  (* donja fizicka vrednost opsega [bar] *)
PG.Sens.Pt._NS2.AI_Param.ScaledMax          := 0.3;   (* gornja fizicka vrednost opsega [bar] *)
PG.Sens.Pt._NS2.AI_Param.UnitOfMeasure      := 'bar';  (* jedinica za prikaz na HMI *)
PG.Sens.Pt._NS2.AI_Param.EnableStatusCheck  := FALSE;   (* bez TransmitterStatus DI - nije prikljucen *)

(* -------------------------------------------------------------------------- *)
(* 3) FBAI01_DI01  Temperature TT_PG_01..TT_PG_07                             *)
(* TT_PG_01..03 su na X20AI4622b, a TT_PG_04..07 na X67AI1323/X67AI1333b.     *)
(* Easytemp TMR35, 4-20mA. Opseg: 0-120 degC.                                  *)
(* -------------------------------------------------------------------------- *)
(* Tt._1 / TT_PG_01: Ulaz u veliki razmenjivac PGRT01 [degC]. *)
PG.Sens.Tt._1.AI_Input.Enable             := TRUE;      (* Aktivira obradu mapiranog AI signala. *)
PG.Sens.Tt._1.AI_Param.RawMin             := 0;         (* 4 mA. *)
PG.Sens.Tt._1.AI_Param.RawMax             := 32767;     (* 20 mA. *)
PG.Sens.Tt._1.AI_Param.ScaledMin          := 0.0;       (* Donja granica [degC]. *)
PG.Sens.Tt._1.AI_Param.ScaledMax          := 120.0;     (* Gornja granica [degC]. *)
PG.Sens.Tt._1.AI_Param.UnitOfMeasure      := 'degC';    (* HMI jedinica. *)
PG.Sens.Tt._1.AI_Param.EnableStatusCheck  := FALSE;     (* Nema statusnog DI signala. *)

(* Tt._2 / TT_PG_02: Temperatura na ulazu u prihvatni tank [degC]. *)
PG.Sens.Tt._2.AI_Input.Enable             := TRUE;      (* Aktivira obradu mapiranog AI signala. *)
PG.Sens.Tt._2.AI_Param.RawMin             := 0;         (* 4 mA. *)
PG.Sens.Tt._2.AI_Param.RawMax             := 32767;     (* 20 mA. *)
PG.Sens.Tt._2.AI_Param.ScaledMin          := 0.0;       (* Donja granica [degC]. *)
PG.Sens.Tt._2.AI_Param.ScaledMax          := 120.0;     (* Gornja granica [degC]. *)
PG.Sens.Tt._2.AI_Param.UnitOfMeasure      := 'degC';    (* HMI jedinica. *)
PG.Sens.Tt._2.AI_Param.EnableStatusCheck  := FALSE;     (* Nema statusnog DI signala. *)

(* Tt._3 / TT_PG_03: Temperatura u prihvatnom tanku [degC]. *)
PG.Sens.Tt._3.AI_Input.Enable             := TRUE;      (* Aktivira obradu mapiranog AI signala. *)
PG.Sens.Tt._3.AI_Param.RawMin             := 0;         (* 4 mA. *)
PG.Sens.Tt._3.AI_Param.RawMax             := 32767;     (* 20 mA. *)
PG.Sens.Tt._3.AI_Param.ScaledMin          := 0.0;       (* Donja granica [degC]. *)
PG.Sens.Tt._3.AI_Param.ScaledMax          := 120.0;     (* Gornja granica [degC]. *)
PG.Sens.Tt._3.AI_Param.UnitOfMeasure      := 'degC';    (* HMI jedinica. *)
PG.Sens.Tt._3.AI_Param.EnableStatusCheck  := FALSE;     (* Nema statusnog DI signala. *)

(* Tt._4 / TT_PG_04: Izlaz iz velikog razmenjivaca PGRT01 [degC]. *)
PG.Sens.Tt._4.AI_Input.Enable             := TRUE;      (* Aktivira obradu mapiranog AI signala. *)
PG.Sens.Tt._4.AI_Param.RawMin             := 0;         (* 4 mA. *)
PG.Sens.Tt._4.AI_Param.RawMax             := 32767;     (* 20 mA. *)
PG.Sens.Tt._4.AI_Param.ScaledMin          := 0.0;       (* Donja granica [degC]. *)
PG.Sens.Tt._4.AI_Param.ScaledMax          := 120.0;     (* Gornja granica [degC]. *)
PG.Sens.Tt._4.AI_Param.UnitOfMeasure      := 'degC';    (* HMI jedinica. *)
PG.Sens.Tt._4.AI_Param.EnableStatusCheck  := FALSE;     (* Nema statusnog DI signala. *)

(* Tt._5 / TT_PG_05: Ulaz u mali razmenjivac PGRT02 [degC]. *)
PG.Sens.Tt._5.AI_Input.Enable             := TRUE;      (* Aktivira obradu mapiranog AI signala. *)
PG.Sens.Tt._5.AI_Param.RawMin             := 0;         (* 4 mA. *)
PG.Sens.Tt._5.AI_Param.RawMax             := 32767;     (* 20 mA. *)
PG.Sens.Tt._5.AI_Param.ScaledMin          := 0.0;       (* Donja granica [degC]. *)
PG.Sens.Tt._5.AI_Param.ScaledMax          := 120.0;     (* Gornja granica [degC]. *)
PG.Sens.Tt._5.AI_Param.UnitOfMeasure      := 'degC';    (* HMI jedinica. *)
PG.Sens.Tt._5.AI_Param.EnableStatusCheck  := FALSE;     (* Nema statusnog DI signala. *)

(* Tt._6 / TT_PG_06: Izlaz iz malog razmenjivaca PGRT02 [degC]. *)
PG.Sens.Tt._6.AI_Input.Enable             := TRUE;      (* Aktivira obradu mapiranog AI signala. *)
PG.Sens.Tt._6.AI_Param.RawMin             := 0;         (* 4 mA. *)
PG.Sens.Tt._6.AI_Param.RawMax             := 32767;     (* 20 mA. *)
PG.Sens.Tt._6.AI_Param.ScaledMin          := 0.0;       (* Donja granica [degC]. *)
PG.Sens.Tt._6.AI_Param.ScaledMax          := 120.0;     (* Gornja granica [degC]. *)
PG.Sens.Tt._6.AI_Param.UnitOfMeasure      := 'degC';    (* HMI jedinica. *)
PG.Sens.Tt._6.AI_Param.EnableStatusCheck  := FALSE;     (* Nema statusnog DI signala. *)

(* Tt._7 / TT_PG_07: Drenazni vod za potvrdu zavrsetka preispiranja [degC]. *)
PG.Sens.Tt._7.AI_Input.Enable             := TRUE;      (* Aktivira obradu mapiranog AI signala. *)
PG.Sens.Tt._7.AI_Param.RawMin             := 0;         (* 4 mA. *)
PG.Sens.Tt._7.AI_Param.RawMax             := 32767;     (* 20 mA. *)
PG.Sens.Tt._7.AI_Param.ScaledMin          := 0.0;       (* Donja granica [degC]. *)
PG.Sens.Tt._7.AI_Param.ScaledMax          := 120.0;     (* Gornja granica [degC]. *)
PG.Sens.Tt._7.AI_Param.UnitOfMeasure      := 'degC';    (* HMI jedinica. *)
PG.Sens.Tt._7.AI_Param.EnableStatusCheck  := FALSE;     (* Nema statusnog DI signala. *)

(* -------------------------------------------------------------------------- *)
(* 3.1) FBAI01_DI01  Temperature TT_PG_08..TT_PG_11                        *)
(* Tehnicka i sanitarna voda kroz direktni izmenjivac, 0..120 degC.          *)
(* -------------------------------------------------------------------------- *)
(* Tt._8 / TT_PG_08: ulaz tehnicke vode u direktni izmenjivac [degC]. *)
PG.Sens.Tt._8.AI_Input.Enable             := TRUE;      (* Aktivira obradu mapiranog AI signala. *)
PG.Sens.Tt._8.AI_Param.RawMin             := 0;         (* 4 mA. *)
PG.Sens.Tt._8.AI_Param.RawMax             := 32767;     (* 20 mA. *)
PG.Sens.Tt._8.AI_Param.ScaledMin          := 0.0;       (* Donja granica [degC]. *)
PG.Sens.Tt._8.AI_Param.ScaledMax          := 120.0;     (* Gornja granica [degC]. *)
PG.Sens.Tt._8.AI_Param.UnitOfMeasure      := 'degC';    (* HMI jedinica. *)
PG.Sens.Tt._8.AI_Param.EnableStatusCheck  := FALSE;     (* Nema statusnog DI signala. *)

(* Tt._9 / TT_PG_09: izlaz tehnicke vode iz direktnog izmenjivaca [degC]. *)
PG.Sens.Tt._9.AI_Input.Enable             := TRUE;      (* Aktivira obradu mapiranog AI signala. *)
PG.Sens.Tt._9.AI_Param.RawMin             := 0;         (* 4 mA. *)
PG.Sens.Tt._9.AI_Param.RawMax             := 32767;     (* 20 mA. *)
PG.Sens.Tt._9.AI_Param.ScaledMin          := 0.0;       (* Donja granica [degC]. *)
PG.Sens.Tt._9.AI_Param.ScaledMax          := 120.0;     (* Gornja granica [degC]. *)
PG.Sens.Tt._9.AI_Param.UnitOfMeasure      := 'degC';    (* HMI jedinica. *)
PG.Sens.Tt._9.AI_Param.EnableStatusCheck  := FALSE;     (* Nema statusnog DI signala. *)

(* Tt._10 / TT_PG_10: ulaz sanitarne vode u direktni izmenjivac [degC]. *)
PG.Sens.Tt._10.AI_Input.Enable            := TRUE;      (* Aktivira obradu mapiranog AI signala. *)
PG.Sens.Tt._10.AI_Param.RawMin            := 0;         (* 4 mA. *)
PG.Sens.Tt._10.AI_Param.RawMax            := 32767;     (* 20 mA. *)
PG.Sens.Tt._10.AI_Param.ScaledMin         := 0.0;       (* Donja granica [degC]. *)
PG.Sens.Tt._10.AI_Param.ScaledMax         := 120.0;     (* Gornja granica [degC]. *)
PG.Sens.Tt._10.AI_Param.UnitOfMeasure     := 'degC';    (* HMI jedinica. *)
PG.Sens.Tt._10.AI_Param.EnableStatusCheck := FALSE;     (* Nema statusnog DI signala. *)

(* Tt._11 / TT_PG_11: izlaz sanitarne vode iz direktnog izmenjivaca [degC]. *)
PG.Sens.Tt._11.AI_Input.Enable            := TRUE;      (* Aktivira obradu mapiranog AI signala. *)
PG.Sens.Tt._11.AI_Param.RawMin            := 0;         (* 4 mA. *)
PG.Sens.Tt._11.AI_Param.RawMax            := 32767;     (* 20 mA. *)
PG.Sens.Tt._11.AI_Param.ScaledMin         := 0.0;       (* Donja granica [degC]. *)
PG.Sens.Tt._11.AI_Param.ScaledMax         := 120.0;     (* Gornja granica [degC]. *)
PG.Sens.Tt._11.AI_Param.UnitOfMeasure     := 'degC';    (* HMI jedinica. *)
PG.Sens.Tt._11.AI_Param.EnableStatusCheck := FALSE;     (* Nema statusnog DI signala. *)

(* -------------------------------------------------------------------------- *)
(* 4) FBAI01_DI01  Merac protoka MP (_1)                                      *)
(* X20AI4622c AI01, 4-20mA, Promag H10 DN065. Opseg: 0-10 l/s.                *)
(* EnableStatusCheck=TRUE: TransmitterStatus DI mapiran u IoMap.              *)
(* -------------------------------------------------------------------------- *)
(* MP._1: Merac protoka na potisu tople termalne vode ka potrosacima [m3/h]  *)
PG.Sens.MP._1.AI_Input.Enable             := TRUE;      (* aktivira FB, pokrece skaliranje i statusnu logiku *)
PG.Sens.MP._1.AI_Param.RawMin             := 0;         (* donja granica raw ADC opsega (0 = 4mA) *)
PG.Sens.MP._1.AI_Param.RawMax             := 32767;     (* gornja granica raw ADC opsega (32767 = 20mA) *)
PG.Sens.MP._1.AI_Param.ScaledMin          := 0.0;       (* min protok [m3/h], 0 l/s *)
PG.Sens.MP._1.AI_Param.ScaledMax          := 20.0;      (* max protok [m3/h], 20 l/s *)
PG.Sens.MP._1.AI_Param.UnitOfMeasure      := 'l/s';    (* jedinica za prikaz na HMI *)
PG.Sens.MP._1.AI_Param.EnableStatusCheck  := TRUE;      (* Promag H10 status DI aktivan, mapiran u IoMap *)

(* -------------------------------------------------------------------------- *)
(* 5) FB_DI  Nivo prekidaci LS (_1.._5)                                       *)
(* Liquipoint FTW23, Tri clamp DN040: detekcija prisustva tecnosti u odzraci. *)
(* DelayOn/Off=T#1s za filtriranje kratkih tranzijenta.                       *)
(* -------------------------------------------------------------------------- *)
(* LS._1: Nizak nivo vode u prihvatnom tanku za rad pumpi *)
PG.Sens.LS._1.DI_Input.Enable          := TRUE;         (* aktivira FB pracenja DI signala *)
PG.Sens.LS._1.DI_Param.UseStatusInput  := FALSE;        (* nema poseban DI za status uredaja *)
PG.Sens.LS._1.DI_Param.InvertSignal    := FALSE;        (* signal se NE invertuje *)
PG.Sens.LS._1.DI_Param.DelayOn         := T#1s;         (* kasnjenje aktivacije - filtriranje tranzijenta *)
PG.Sens.LS._1.DI_Param.DelayOff        := T#1s;         (* kasnjenje deaktivacije - filtriranje tranzijenta *)
PG.Sens.LS._1.DI_Param.TextTrue        := 'Tecnost prisutna';  (* tekst za HMI kada je DI aktivan *)
PG.Sens.LS._1.DI_Param.TextFalse       := 'Tecnost odsutna';   (* tekst za HMI kada je DI neaktivan *)
PG.Sens.LS._1.DI_Param.TextAlarm       := 'LS alarm';   (* tekst alarma za HMI i logovanje *)
PG.Sens.LS._1.DI_Param.TextFault       := 'LS fault';   (* tekst kvara za HMI i logovanje *)

(* LS._2: Donji nivo u odzracnom cilindru na ulazu vode u podstanicu *)
PG.Sens.LS._2.DI_Input.Enable          := TRUE;         (* aktivira FB pracenja DI signala *)
PG.Sens.LS._2.DI_Param.UseStatusInput  := FALSE;        (* nema poseban DI za status uredaja *)
PG.Sens.LS._2.DI_Param.InvertSignal    := FALSE;        (* signal se NE invertuje *)
PG.Sens.LS._2.DI_Param.DelayOn         := T#1s;         (* kasnjenje aktivacije - filtriranje tranzijenta *)
PG.Sens.LS._2.DI_Param.DelayOff        := T#1s;         (* kasnjenje deaktivacije - filtriranje tranzijenta *)
PG.Sens.LS._2.DI_Param.TextTrue        := 'Tecnost prisutna';  (* tekst za HMI kada je DI aktivan *)
PG.Sens.LS._2.DI_Param.TextFalse       := 'Tecnost odsutna';   (* tekst za HMI kada je DI neaktivan *)
PG.Sens.LS._2.DI_Param.TextAlarm       := 'LS alarm';   (* tekst alarma za HMI i logovanje *)
PG.Sens.LS._2.DI_Param.TextFault       := 'LS fault';   (* tekst kvara za HMI i logovanje *)

(* LS._3: Gornji nivo u odzracnom cilindru na ulazu vode u podstanicu *)
PG.Sens.LS._3.DI_Input.Enable          := TRUE;         (* aktivira FB pracenja DI signala *)
PG.Sens.LS._3.DI_Param.UseStatusInput  := FALSE;        (* nema poseban DI za status uredaja *)
PG.Sens.LS._3.DI_Param.InvertSignal    := FALSE;        (* signal se NE invertuje *)
PG.Sens.LS._3.DI_Param.DelayOn         := T#1s;         (* kasnjenje aktivacije - filtriranje tranzijenta *)
PG.Sens.LS._3.DI_Param.DelayOff        := T#1s;         (* kasnjenje deaktivacije - filtriranje tranzijenta *)
PG.Sens.LS._3.DI_Param.TextTrue        := 'Tecnost prisutna';  (* tekst za HMI kada je DI aktivan *)
PG.Sens.LS._3.DI_Param.TextFalse       := 'Tecnost odsutna';   (* tekst za HMI kada je DI neaktivan *)
PG.Sens.LS._3.DI_Param.TextAlarm       := 'LS alarm';   (* tekst alarma za HMI i logovanje *)
PG.Sens.LS._3.DI_Param.TextFault       := 'LS fault';   (* tekst kvara za HMI i logovanje *)

(* LS._4: Donji nivo u odzracnom cilindru na ulazu vode u prihvatni tank *)
PG.Sens.LS._4.DI_Input.Enable          := TRUE;         (* aktivira FB pracenja DI signala *)
PG.Sens.LS._4.DI_Param.UseStatusInput  := FALSE;        (* nema poseban DI za status uredaja *)
PG.Sens.LS._4.DI_Param.InvertSignal    := FALSE;        (* signal se NE invertuje *)
PG.Sens.LS._4.DI_Param.DelayOn         := T#1s;         (* kasnjenje aktivacije - filtriranje tranzijenta *)
PG.Sens.LS._4.DI_Param.DelayOff        := T#1s;         (* kasnjenje deaktivacije - filtriranje tranzijenta *)
PG.Sens.LS._4.DI_Param.TextTrue        := 'Tecnost prisutna';  (* tekst za HMI kada je DI aktivan *)
PG.Sens.LS._4.DI_Param.TextFalse       := 'Tecnost odsutna';   (* tekst za HMI kada je DI neaktivan *)
PG.Sens.LS._4.DI_Param.TextAlarm       := 'LS alarm';   (* tekst alarma za HMI i logovanje *)
PG.Sens.LS._4.DI_Param.TextFault       := 'LS fault';   (* tekst kvara za HMI i logovanje *)

(* LS._5: Gornji nivo u odzracnom cilindru na ulazu vode u prihvatni tank *)
PG.Sens.LS._5.DI_Input.Enable          := TRUE;         (* aktivira FB pracenja DI signala *)
PG.Sens.LS._5.DI_Param.UseStatusInput  := FALSE;        (* nema poseban DI za status uredaja *)
PG.Sens.LS._5.DI_Param.InvertSignal    := FALSE;        (* signal se NE invertuje *)
PG.Sens.LS._5.DI_Param.DelayOn         := T#1s;         (* kasnjenje aktivacije - filtriranje tranzijenta *)
PG.Sens.LS._5.DI_Param.DelayOff        := T#1s;         (* kasnjenje deaktivacije - filtriranje tranzijenta *)
PG.Sens.LS._5.DI_Param.TextTrue        := 'Tecnost prisutna';  (* tekst za HMI kada je DI aktivan *)
PG.Sens.LS._5.DI_Param.TextFalse       := 'Tecnost odsutna';   (* tekst za HMI kada je DI neaktivan *)
PG.Sens.LS._5.DI_Param.TextAlarm       := 'LS alarm';   (* tekst alarma za HMI i logovanje *)
PG.Sens.LS._5.DI_Param.TextFault       := 'LS fault';   (* tekst kvara za HMI i logovanje *)

(* -------------------------------------------------------------------------- *)
(* 6) FB_DI  Prestrujni ventili OWF (_1, _2)                                  *)
(* NIOB FLUID 5371 DN050, povratni signal otvorenog polozaja 3-5 bara.        *)
(* DelayOn/Off=T#500ms za filtriranje kratkih tranzijenta pri promeni pritiska.*)
(* -------------------------------------------------------------------------- *)
(* OWF._1: Zastitni prestrujni ventil od hidraulickog udara 1 *)
PG.Sens.OWF._1.DI_Input.Enable          := TRUE;        (* aktivira FB pracenja DI signala *)
PG.Sens.OWF._1.DI_Param.UseStatusInput  := FALSE;       (* nema poseban DI za status uredaja *)
PG.Sens.OWF._1.DI_Param.InvertSignal    := FALSE;       (* signal se NE invertuje *)
PG.Sens.OWF._1.DI_Param.DelayOn         := T#500ms;     (* kasnjenje aktivacije - filtriranje pri promeni pritiska *)
PG.Sens.OWF._1.DI_Param.DelayOff        := T#500ms;     (* kasnjenje deaktivacije - filtriranje pri promeni pritiska *)
PG.Sens.OWF._1.DI_Param.TextTrue        := 'OWF otvoren';   (* tekst za HMI kada je ventil otvoren *)
PG.Sens.OWF._1.DI_Param.TextFalse       := 'OWF zatvoren';  (* tekst za HMI kada je ventil zatvoren *)
PG.Sens.OWF._1.DI_Param.TextAlarm       := 'OWF alarm';     (* tekst alarma za HMI i logovanje *)
PG.Sens.OWF._1.DI_Param.TextFault       := 'OWF fault';     (* tekst kvara za HMI i logovanje *)

(* OWF._2: Zastitni prestrujni ventil od hidraulickog udara 2 *)
PG.Sens.OWF._2.DI_Input.Enable          := TRUE;        (* aktivira FB pracenja DI signala *)
PG.Sens.OWF._2.DI_Param.UseStatusInput  := FALSE;       (* nema poseban DI za status uredaja *)
PG.Sens.OWF._2.DI_Param.InvertSignal    := FALSE;       (* signal se NE invertuje *)
PG.Sens.OWF._2.DI_Param.DelayOn         := T#500ms;     (* kasnjenje aktivacije - filtriranje pri promeni pritiska *)
PG.Sens.OWF._2.DI_Param.DelayOff        := T#500ms;     (* kasnjenje deaktivacije - filtriranje pri promeni pritiska *)
PG.Sens.OWF._2.DI_Param.TextTrue        := 'OWF otvoren';   (* tekst za HMI kada je ventil otvoren *)
PG.Sens.OWF._2.DI_Param.TextFalse       := 'OWF zatvoren';  (* tekst za HMI kada je ventil zatvoren *)
PG.Sens.OWF._2.DI_Param.TextAlarm       := 'OWF alarm';     (* tekst alarma za HMI i logovanje *)
PG.Sens.OWF._2.DI_Param.TextFault       := 'OWF fault';     (* tekst kvara za HMI i logovanje *)

(* -------------------------------------------------------------------------- *)
(* 7) FB_V_EMV + FB_V_ON_OFF_FB  Automatski ventili AV (_1.._7)               *)
(* AV._1, _2: End Armaturen DN125, elektromotorni bistabilni, CmdOpen+CmdClose*)
(* AV._3.._7: End Armaturen DN125, pneumatski NC spring-return, samo Cmd.     *)
(* OpenMaxTime: bistabilni=20s, spring-return=10s.                             *)
(* AV._1/_2 koriste PositionConfirmTime; AV._3.._7 koriste StableFbDelay.     *)
(* -------------------------------------------------------------------------- *)
(* AV._1: Elektromotorni leptir ventil DN125 bistabilan  razmenjivac toplote *)
PG.Act.AV._1.V_Input.Enable            := FALSE;         (* aktivira FB upravljanja ventilom *)
PG.Act.AV._1.V_Input.ForceCmd      	   := FALSE;         (* komanda ide na izlaz bez obzira na stanje / alarm *)
PG.Act.AV._1.V_Param.LampOpenExists    := TRUE;         (* pomocni DI signal LampOpen je dostupan i koristi se u logici FB-a *)
PG.Act.AV._1.V_Param.LampCloseExists   := TRUE;         (* pomocni DI signal LampClose je dostupan i koristi se u logici FB-a *)
PG.Act.AV._1.V_Param.OpenFbExists      := TRUE;         (* postoji DI povratni signal za otvoreni polozaj *)
PG.Act.AV._1.V_Param.CloseFbExists     := TRUE;         (* postoji DI povratni signal za zatvoreni polozaj *)
PG.Act.AV._1.V_Param.OverTorqueExists  := TRUE;         (* postoji DI signal preopterecenja za AV._1 *)
PG.Act.AV._1.V_Param.OpenMaxTime       := T#20s;        (* timeout - alarm ako FB otvoren ne stigne za 20s *)
PG.Act.AV._1.V_Param.CloseMaxTime      := T#20s;        (* timeout - alarm ako FB zatvoren ne stigne za 20s *)
PG.Act.AV._1.V_Param.EndLimitFilterTime := T#50ms;      (* filtriranje LampOpen/LampClose signala pre evaluacije stanja *)
PG.Act.AV._1.V_Param.PositionFbFilterTime := T#100ms;   (* filtriranje OpenFb/CloseFb signala pre potvrde pozicije *)
PG.Act.AV._1.V_Param.OverTorqueFilterTime := T#20ms;    (* filtriranje preopterecenja pre formiranja fault uslova *)
PG.Act.AV._1.V_Param.PositionConfirmTime := T#2s;       (* vreme cekanja trajnog feedback-a nakon krajnjeg polozaja *)

(* AV._2: Elektromotorni leptir ventil DN125 bistabilan  razmenjivac toplote *)
PG.Act.AV._2.V_Input.Enable            := FALSE;         (* aktivira FB upravljanja ventilom *)
PG.Act.AV._2.V_Input.ForceCmd      	   := FALSE;         (* komanda ide na izlaz bez obzira na stanje / alarm *)
PG.Act.AV._2.V_Param.LampOpenExists    := TRUE;         (* pomocni DI signal LampOpen je dostupan i koristi se u logici FB-a *)
PG.Act.AV._2.V_Param.LampCloseExists   := TRUE;         (* pomocni DI signal LampClose je dostupan i koristi se u logici FB-a *)
PG.Act.AV._2.V_Param.OpenFbExists      := TRUE;         (* postoji DI povratni signal za otvoreni polozaj *)
PG.Act.AV._2.V_Param.CloseFbExists     := TRUE;         (* postoji DI povratni signal za zatvoreni polozaj *)
PG.Act.AV._2.V_Param.OverTorqueExists  := FALSE;        (* AV._2 nema fizicki DI signal preopterecenja *)
PG.Act.AV._2.V_Param.OpenMaxTime       := T#20s;        (* timeout - alarm ako FB otvoren ne stigne za 20s *)
PG.Act.AV._2.V_Param.CloseMaxTime      := T#20s;        (* timeout - alarm ako FB zatvoren ne stigne za 20s *)
PG.Act.AV._2.V_Param.EndLimitFilterTime := T#50ms;      (* filtriranje LampOpen/LampClose signala pre evaluacije stanja *)
PG.Act.AV._2.V_Param.PositionFbFilterTime := T#100ms;   (* filtriranje OpenFb/CloseFb signala pre potvrde pozicije *)
PG.Act.AV._2.V_Param.PositionConfirmTime := T#2s;       (* vreme cekanja trajnog feedback-a nakon krajnjeg polozaja *)

(* AV._3: Pneumatski NC leptir ventil DN125 spring-return  prihvatni tank 1 *)
PG.Act.AV._3.V_Input.Enable            := TRUE;         (* aktivira FB upravljanja ventilom *)
PG.Act.AV._3.V_Input.ForceCmd      	   := TRUE;         (* komanda ide na izlaz bez obzira na stanje / alarm *)
PG.Act.AV._3.V_Param.FbOpenExists      := TRUE;         (* postoji DI povratni signal za otvoreni polozaj *)
PG.Act.AV._3.V_Param.FbCloseExists     := TRUE;         (* postoji DI povratni signal za zatvoreni polozaj *)
PG.Act.AV._3.V_Param.OpenMinTime       := T#0s;         (* min vreme drzanja komande otvori pre provere FB *)
PG.Act.AV._3.V_Param.OpenMaxTime       := T#10s;        (* timeout - spring-return brzi od elektromotornog *)
PG.Act.AV._3.V_Param.CloseMinTime      := T#0s;         (* min vreme drzanja komande zatvori pre provere FB *)
PG.Act.AV._3.V_Param.CloseMaxTime      := T#10s;        (* timeout - spring-return brzi od elektromotornog *)
PG.Act.AV._3.V_Param.StableFbDelay     := T#2s;         (* vreme stabilizacije FB signala pre potvrde polozaja *)

(* AV._4: Pneumatski NC leptir ventil DN125 spring-return  prihvatni tank 2 *)
PG.Act.AV._4.V_Input.Enable            := TRUE;         (* aktivira FB upravljanja ventilom *)
PG.Act.AV._4.V_Input.ForceCmd      	   := TRUE;         (* komanda ide na izlaz bez obzira na stanje / alarm *)
PG.Act.AV._4.V_Param.FbOpenExists      := TRUE;         (* postoji DI povratni signal za otvoreni polozaj *)
PG.Act.AV._4.V_Param.FbCloseExists     := TRUE;         (* postoji DI povratni signal za zatvoreni polozaj *)
PG.Act.AV._4.V_Param.OpenMinTime       := T#0s;         (* min vreme drzanja komande otvori pre provere FB *)
PG.Act.AV._4.V_Param.OpenMaxTime       := T#10s;        (* timeout - spring-return brzi od elektromotornog *)
PG.Act.AV._4.V_Param.CloseMinTime      := T#0s;         (* min vreme drzanja komande zatvori pre provere FB *)
PG.Act.AV._4.V_Param.CloseMaxTime      := T#10s;        (* timeout - spring-return brzi od elektromotornog *)
PG.Act.AV._4.V_Param.StableFbDelay     := T#2s;         (* vreme stabilizacije FB signala pre potvrde polozaja *)

(* AV._5: Pneumatski NC leptir ventil DN125 spring-return *)
PG.Act.AV._5.V_Input.Enable            := TRUE;         (* aktivira FB upravljanja ventilom *)
PG.Act.AV._5.V_Input.ForceCmd      	   := TRUE;         (* komanda ide na izlaz bez obzira na stanje / alarm *)
PG.Act.AV._5.V_Param.FbOpenExists      := TRUE;         (* postoji DI povratni signal za otvoreni polozaj *)
PG.Act.AV._5.V_Param.FbCloseExists     := TRUE;         (* postoji DI povratni signal za zatvoreni polozaj *)
PG.Act.AV._5.V_Param.OpenMinTime       := T#0s;         (* min vreme drzanja komande otvori pre provere FB *)
PG.Act.AV._5.V_Param.OpenMaxTime       := T#10s;        (* timeout - spring-return brzi od elektromotornog *)
PG.Act.AV._5.V_Param.CloseMinTime      := T#0s;         (* min vreme drzanja komande zatvori pre provere FB *)
PG.Act.AV._5.V_Param.CloseMaxTime      := T#10s;        (* timeout - spring-return brzi od elektromotornog *)
PG.Act.AV._5.V_Param.StableFbDelay     := T#2s;         (* vreme stabilizacije FB signala pre potvrde polozaja *)

(* AV._6: Pneumatski NC leptir ventil DN125 spring-return *)
PG.Act.AV._6.V_Input.Enable            := TRUE;         (* aktivira FB upravljanja ventilom *)
PG.Act.AV._6.V_Input.ForceCmd      	   := TRUE;         (* komanda ide na izlaz bez obzira na stanje / alarm *)
PG.Act.AV._6.V_Param.FbOpenExists      := TRUE;         (* postoji DI povratni signal za otvoreni polozaj *)
PG.Act.AV._6.V_Param.FbCloseExists     := TRUE;         (* postoji DI povratni signal za zatvoreni polozaj *)
PG.Act.AV._6.V_Param.OpenMinTime       := T#0s;         (* min vreme drzanja komande otvori pre provere FB *)
PG.Act.AV._6.V_Param.OpenMaxTime       := T#10s;        (* timeout - spring-return brzi od elektromotornog *)
PG.Act.AV._6.V_Param.CloseMinTime      := T#0s;         (* min vreme drzanja komande zatvori pre provere FB *)
PG.Act.AV._6.V_Param.CloseMaxTime      := T#10s;        (* timeout - spring-return brzi od elektromotornog *)
PG.Act.AV._6.V_Param.StableFbDelay     := T#2s;         (* vreme stabilizacije FB signala pre potvrde polozaja *)

(* AV._7: Pneumatski NC leptir ventil DN125 spring-return *)
PG.Act.AV._7.V_Input.Enable            := TRUE;         (* aktivira FB upravljanja ventilom *)
PG.Act.AV._7.V_Input.ForceCmd      	   := TRUE;         (* komanda ide na izlaz bez obzira na stanje / alarm *)
PG.Act.AV._7.V_Param.FbOpenExists      := TRUE;         (* postoji DI povratni signal za otvoreni polozaj *)
PG.Act.AV._7.V_Param.FbCloseExists     := TRUE;         (* postoji DI povratni signal za zatvoreni polozaj *)
PG.Act.AV._7.V_Param.OpenMinTime       := T#0s;         (* min vreme drzanja komande otvori pre provere FB *)
PG.Act.AV._7.V_Param.OpenMaxTime       := T#10s;        (* timeout - spring-return brzi od elektromotornog *)
PG.Act.AV._7.V_Param.CloseMinTime      := T#0s;         (* min vreme drzanja komande zatvori pre provere FB *)
PG.Act.AV._7.V_Param.CloseMaxTime      := T#10s;        (* timeout - spring-return brzi od elektromotornog *)
PG.Act.AV._7.V_Param.StableFbDelay     := T#2s;         (* vreme stabilizacije FB signala pre potvrde polozaja *)

(* -------------------------------------------------------------------------- *)
(* 8) FB_HV_2LS  Rucni leptir ventili RV (_19, _21.._27)                      *)
(* NIOB FLUID 4309 / End Armaturen, rucni C-C sa povratnim signalima.         *)
(* TransitionMaxTime=T#10s: alarm ako tranzicija prekoraci 10s.               *)
(* BothActiveFilterTime=T#500ms: debounce oba krajnja signala.                *)
(* -------------------------------------------------------------------------- *)
(* RV._19: Rucni ventil posle membranskog ventila PG_PV01 *)
PG.Act.RV._19.HV_Input.Enable          := TRUE;         (* aktivira FB monitoringa rucnog ventila *)
PG.Act.RV._19.HV_Param.TransitionMaxTime := T#10s;      (* timeout alarm pri tranziciji polozaja *)
PG.Act.RV._19.HV_Param.BothActiveFilterTime := T#500ms; (* debounce za oba FB aktivna istovremeno *)

(* RV._21: Rucni ventil posle membranskog ventila PG_PV02 *)
PG.Act.RV._21.HV_Input.Enable          := TRUE;         (* aktivira FB monitoringa rucnog ventila *)
PG.Act.RV._21.HV_Param.TransitionMaxTime := T#10s;      (* timeout alarm pri tranziciji polozaja *)
PG.Act.RV._21.HV_Param.BothActiveFilterTime := T#500ms; (* debounce za oba FB aktivna istovremeno *)

(* RV._22: Drenazni total ventil na dnu prihvatnog tanka *)
PG.Act.RV._22.HV_Input.Enable          := TRUE;         (* aktivira FB monitoringa rucnog ventila *)
PG.Act.RV._22.HV_Param.TransitionMaxTime := T#10s;      (* timeout alarm pri tranziciji polozaja *)
PG.Act.RV._22.HV_Param.BothActiveFilterTime := T#500ms; (* debounce za oba FB aktivna istovremeno *)

(* RV._23: Ulaz u Pumpu PG_Pu01 *)
PG.Act.RV._23.HV_Input.Enable          := TRUE;         (* aktivira FB monitoringa rucnog ventila *)
PG.Act.RV._23.HV_Param.TransitionMaxTime := T#10s;      (* timeout alarm pri tranziciji polozaja *)
PG.Act.RV._23.HV_Param.BothActiveFilterTime := T#500ms; (* debounce za oba FB aktivna istovremeno *)

(* RV._24: Ulaz u Pumpu PG_Pu02 *)
PG.Act.RV._24.HV_Input.Enable          := TRUE;         (* aktivira FB monitoringa rucnog ventila *)
PG.Act.RV._24.HV_Param.TransitionMaxTime := T#10s;      (* timeout alarm pri tranziciji polozaja *)
PG.Act.RV._24.HV_Param.BothActiveFilterTime := T#500ms; (* debounce za oba FB aktivna istovremeno *)

(* RV._25: Bajpasni izlaz iz tanka ka instalaciji za izbacivanje gasa van kotlarnice *)
PG.Act.RV._25.HV_Input.Enable          := TRUE;         (* aktivira FB monitoringa rucnog ventila *)
PG.Act.RV._25.HV_Param.TransitionMaxTime := T#10s;      (* timeout alarm pri tranziciji polozaja *)
PG.Act.RV._25.HV_Param.BothActiveFilterTime := T#500ms; (* debounce za oba FB aktivna istovremeno *)

(* RV._26: Ulaz u vakuum pumpu *)
PG.Act.RV._26.HV_Input.Enable          := TRUE;         (* aktivira FB monitoringa rucnog ventila *)
PG.Act.RV._26.HV_Param.TransitionMaxTime := T#10s;      (* timeout alarm pri tranziciji polozaja *)
PG.Act.RV._26.HV_Param.BothActiveFilterTime := T#500ms; (* debounce za oba FB aktivna istovremeno *)

(* RV._27: Izlaz iz vakuum pumpe ka instalaciji za izbacivanje gasa van kotlarnice *)
PG.Act.RV._27.HV_Input.Enable          := TRUE;         (* aktivira FB monitoringa rucnog ventila *)
PG.Act.RV._27.HV_Param.TransitionMaxTime := T#10s;      (* timeout alarm pri tranziciji polozaja *)
PG.Act.RV._27.HV_Param.BothActiveFilterTime := T#500ms; (* debounce za oba FB aktivna istovremeno *)

(* -------------------------------------------------------------------------- *)
(* 9) FB_PvAiAo_Fast  Proporcionalni membranski ventili PV (_1.._5)           *)
(* Burkert, AI povratni signal + AO komanda, 4-20mA, mapirano u IoMap.        *)
(* DeviationOnLimit=8%: alarm ako fizicki polozaj odstupa > 8% od SP.         *)
(* DeviationOffLimit=3%: alarm se gasi kada padne ispod 3% odstupanja.        *)
(* -------------------------------------------------------------------------- *)
(* PV._1: Ulazni regulacioni ventil 1 - prihvatni tank, DN050 NC *)
PG.Act.PV._1.PV_Input.Enable               := TRUE;     (* aktivira FB proporc. ventila *)
PG.Act.PV._1.PV_Input.ForceCmd             := TRUE;     (* komanda ide na izlaz bez obzira na stanje / alarm *)
PG.Act.PV._1.PV_Param.HoldOutputOnFault    := TRUE;     (* zadrzava poslednju AO vrednost pri kvar signalu *)
PG.Act.PV._1.PV_Param.DeviationOnLimit     := 8.0;      (* [%] alarm aktivira se kada odstupanje predje 8% *)
PG.Act.PV._1.PV_Param.DeviationOffLimit    := 3.0;      (* [%] alarm gasi se kada odstupanje padne ispod 3% *)
PG.Act.PV._1.PV_Param.DeviationTime        := T#5s;     (* vreme pre aktiviranja alarma odstupanja *)

(* PV._2: Ulazni regulacioni ventil 2 - prihvatni tank, DN050 NC *)
PG.Act.PV._2.PV_Input.Enable               := TRUE;     (* aktivira FB proporc. ventila *)
PG.Act.PV._2.PV_Input.ForceCmd             := TRUE;     (* komanda ide na izlaz bez obzira na stanje / alarm *)
PG.Act.PV._2.PV_Param.HoldOutputOnFault    := TRUE;     (* zadrzava poslednju AO vrednost pri kvar signalu *)
PG.Act.PV._2.PV_Param.DeviationOnLimit     := 8.0;      (* [%] alarm aktivira se kada odstupanje predje 8% *)
PG.Act.PV._2.PV_Param.DeviationOffLimit    := 3.0;      (* [%] alarm gasi se kada odstupanje padne ispod 3% *)
PG.Act.PV._2.PV_Param.DeviationTime        := T#5s;     (* vreme pre aktiviranja alarma odstupanja *)

(* PV._3: Odzracni ventil na ulazu termalne vode u kotlarnicu, DN025 NC *)
PG.Act.PV._3.PV_Input.Enable               := TRUE;     (* aktivira FB proporc. ventila *)
PG.Act.PV._3.PV_Input.ForceCmd             := TRUE;     (* komanda ide na izlaz bez obzira na stanje / alarm *)
PG.Act.PV._3.PV_Param.HoldOutputOnFault    := TRUE;     (* zadrzava poslednju AO vrednost pri kvar signalu *)
PG.Act.PV._3.PV_Param.DeviationOnLimit     := 8.0;      (* [%] alarm aktivira se kada odstupanje predje 8% *)
PG.Act.PV._3.PV_Param.DeviationOffLimit    := 3.0;      (* [%] alarm gasi se kada odstupanje padne ispod 3% *)
PG.Act.PV._3.PV_Param.DeviationTime        := T#5s;     (* vreme pre aktiviranja alarma odstupanja *)

(* PV._4: Odzracni ventil na ulazu termalne vode u prihvatni tank, DN025 NC *)
PG.Act.PV._4.PV_Input.Enable               := TRUE;     (* aktivira FB proporc. ventila *)
PG.Act.PV._4.PV_Input.ForceCmd             := TRUE;     (* komanda ide na izlaz bez obzira na stanje / alarm *)
PG.Act.PV._4.PV_Param.HoldOutputOnFault    := TRUE;     (* zadrzava poslednju AO vrednost pri kvar signalu *)
PG.Act.PV._4.PV_Param.DeviationOnLimit     := 8.0;      (* [%] alarm aktivira se kada odstupanje predje 8% *)
PG.Act.PV._4.PV_Param.DeviationOffLimit    := 3.0;      (* [%] alarm gasi se kada odstupanje padne ispod 3% *)
PG.Act.PV._4.PV_Param.DeviationTime        := T#5s;     (* vreme pre aktiviranja alarma odstupanja *)

(* PV._5: Dodatni proporcionalni ventil, Fast varijanta kao i ostali PV kanali *)
PG.Act.PV._5.PV_Input.Enable               := TRUE;     (* aktivira FB proporc. ventila *)
PG.Act.PV._5.PV_Input.ForceCmd             := TRUE;     (* komanda ide na izlaz bez obzira na stanje / alarm *)
PG.Act.PV._5.PV_Param.HoldOutputOnFault    := TRUE;     (* zadrzava poslednju AO vrednost pri kvar signalu *)
PG.Act.PV._5.PV_Param.DeviationOnLimit     := 8.0;      (* [%] alarm aktivira se kada odstupanje predje 8% *)
PG.Act.PV._5.PV_Param.DeviationOffLimit    := 3.0;      (* [%] alarm gasi se kada odstupanje padne ispod 3% *)
PG.Act.PV._5.PV_Param.DeviationTime        := T#5s;     (* vreme pre aktiviranja alarma odstupanja *)

END_PROGRAM
```

### Program Logical/Project/DeviceCtrl (IEC)

#### Init.st - Init code
```iecst
PROGRAM _INIT
	(* DeviceCtrl koristi parametre inicijalizovane u vlasnickim programima. *)
END_PROGRAM
```

#### Cyclic.st - Cyclic code
```iecst
PROGRAM _CYCLIC
	(* Komande se pripremaju pre nego sto ih IO task prosledi uredjajskim FB-ovima. *)
	CommandMap;
	ValveCtrl;
	PumpCtrl;
	ProcessValues;
END_PROGRAM
```

#### Variables.var - Local variables
```iecst
VAR
	(* HMI impulsi koriguju Pu01 za +1.0/+0.1/-1.0/-0.1 Hz samo kada procesni komandni vektor nije vlasnik. *)
	Pu1_1_plus : BOOL; (* HMI impuls povecanja zahteva PG_Pu01 za 1.0 Hz. *)
	Pu1_01_plus : BOOL; (* HMI impuls povecanja zahteva PG_Pu01 za 0.1 Hz. *)
	Pu1_1_minus : BOOL; (* HMI impuls smanjenja zahteva PG_Pu01 za 1.0 Hz. *)
	Pu1_01_minus : BOOL; (* HMI impuls smanjenja zahteva PG_Pu01 za 0.1 Hz. *)
	(* HMI impulsi koriguju Pu02 za +1.0/+0.1/-1.0/-0.1 Hz samo kada procesni komandni vektor nije vlasnik. *)
	Pu2_1_plus : BOOL; (* HMI impuls povecanja zahteva PG_Pu02 za 1.0 Hz. *)
	Pu2_01_plus : BOOL; (* HMI impuls povecanja zahteva PG_Pu02 za 0.1 Hz. *)
	Pu2_1_minus : BOOL; (* HMI impuls smanjenja zahteva PG_Pu02 za 1.0 Hz. *)
	Pu2_01_minus : BOOL; (* HMI impuls smanjenja zahteva PG_Pu02 za 0.1 Hz. *)
END_VAR
```

#### CommandMap.st
```iecst
ACTION CommandMap:
	(* ======================================================================== *)
	(* COMMANDMAP - VLASNIK FIZICKOG MAPIRANJA                               *)
	(* COMMON: preslikava vec formiran komandni vektor na fizicke izlaze.     *)
	(* AUTO/MANUAL: ne bira rezim; BRB2Rad_Cmd.Aktivan odredjuje vlasnika.    *)
	(* STOP/FAULT: nevalidan ili neaktivan vektor ne prepisuje lokalne izlaze. *)
	(* STATUS: fizicki feedback se obradjuje u IO i alarmnim slojevima.        *)
	(* ======================================================================== *)
	(* ======================================================================== *)
	(* 1) Adapter RETAIN ulaznih ventila                                        *)
	(* ======================================================================== *)
	(* RETAIN vektor je uvek vlasnik komandi V01/V02, nezavisno od procesnog rezima. *)
	PG.Act.AV._1.Open := PGRad.CmdRetain.V01_Open;
	PG.Act.AV._2.Open := PGRad.CmdRetain.V02_Open;

	(* ======================================================================== *)
	(* 2) Adapter neretentivnog upravljackog vektora                            *)
	(* ======================================================================== *)
	(* Ostale komande se prepisuju samo kada je PGRad_Cmd.Aktivan; u suprotnom servisni/lokalni rezim zadrzava ownership. *)
	IF PGRad_Cmd.Aktivan THEN
		PG.Act.AV._3.Open := PGRad_Cmd.Ventili._03_Open;
		PG.Act.AV._4.Open := PGRad_Cmd.Ventili._04_Open;
		PG.Act.AV._5.Open := PGRad_Cmd.Ventili._05_Open;
		PG.Act.AV._6.Open := PGRad_Cmd.Ventili._06_Open;
		PG.Act.AV._7.Open := PGRad_Cmd.Ventili._07_Open;

		PG.Act.PV._1.PV_Input.Enable := PGRad_Cmd.PropVentili.PV01.Enable;
		PG.Act.PV._1.PV_Input.EnableManual := FALSE;
		PG.Act.PV._1.PV_Input.SP_Percent := PGRad_Cmd.PropVentili.PV01.SP_Percent;
		PG.Act.PV._2.PV_Input.Enable := PGRad_Cmd.PropVentili.PV02.Enable;
		PG.Act.PV._2.PV_Input.EnableManual := FALSE;
		PG.Act.PV._2.PV_Input.SP_Percent := PGRad_Cmd.PropVentili.PV02.SP_Percent;
		PG.Act.PV._5.PV_Input.Enable := PGRad_Cmd.PropVentili.PV05.Enable;
		PG.Act.PV._5.PV_Input.EnableManual := FALSE;
		PG.Act.PV._5.PV_Input.SP_Percent := PGRad_Cmd.PropVentili.PV05.SP_Percent;
	END_IF;
END_ACTION
```

#### ValveCtrl.st
```iecst
ACTION ValveCtrl:
	(* ======================================================================== *)
	(* VALVECTRL - PROPORCIONALNI VENTILI I IZLAZNI LIMITI                    *)
	(* AUTO: ProcessUnit/FB_AirRelease daje automatski SP.                    *)
	(* MANUAL: FB manual ulaz se postuje samo kada je lokalni EnableManual TRUE. *)
	(* COMMON: svaki procenat se ogranicava na fizicki opseg 0..100 %.         *)
	(* STOP/FAULT: bez dozvole pripadajuci FB primenjuje svoj bezbedni izlaz.  *)
	(* ======================================================================== *)
	(* ======================================================================== *)
	(* 1) ProcessUnit izlazi odzracnih ventila                                  *)
	(* ======================================================================== *)
	(* ProcessUnit poseduje SP za PV03/PV04; manualni FB ulaz je prisilno iskljucen. *)
	PG.Act.PV._3.PV_Input.EnableManual := FALSE;
	PG.Act.PV._3.PV_Input.SP_Percent := PGRad_AirRelease.PV03.FB.AR_Output.ValveSP_Percent;
	PG.Act.PV._4.PV_Input.EnableManual := FALSE;
	PG.Act.PV._4.PV_Input.SP_Percent := PGRad_AirRelease.PV04.FB.AR_Output.ValveSP_Percent;

	(* ======================================================================== *)
	(* 2) Granice proporcionalnih ventila procesa                               *)
	(* ======================================================================== *)
	(* Clamp 0..100% primenjuje se i na manualnu vrednost i na automatski SP. *)
	IF PG.Act.PV._1.PV_Input.ManualValue_Percent > 100.0 THEN
		PG.Act.PV._1.PV_Input.ManualValue_Percent := 100.0;
	ELSIF PG.Act.PV._1.PV_Input.ManualValue_Percent < 0.0 THEN
		PG.Act.PV._1.PV_Input.ManualValue_Percent := 0.0;
	END_IF;
	IF PG.Act.PV._1.PV_Input.SP_Percent > 100.0 THEN
		PG.Act.PV._1.PV_Input.SP_Percent := 100.0;
	ELSIF PG.Act.PV._1.PV_Input.SP_Percent < 0.0 THEN
		PG.Act.PV._1.PV_Input.SP_Percent := 0.0;
	END_IF;

	IF PG.Act.PV._2.PV_Input.ManualValue_Percent > 100.0 THEN
		PG.Act.PV._2.PV_Input.ManualValue_Percent := 100.0;
	ELSIF PG.Act.PV._2.PV_Input.ManualValue_Percent < 0.0 THEN
		PG.Act.PV._2.PV_Input.ManualValue_Percent := 0.0;
	END_IF;
	IF PG.Act.PV._2.PV_Input.SP_Percent > 100.0 THEN
		PG.Act.PV._2.PV_Input.SP_Percent := 100.0;
	ELSIF PG.Act.PV._2.PV_Input.SP_Percent < 0.0 THEN
		PG.Act.PV._2.PV_Input.SP_Percent := 0.0;
	END_IF;

	IF PG.Act.PV._5.PV_Input.ManualValue_Percent > 100.0 THEN
		PG.Act.PV._5.PV_Input.ManualValue_Percent := 100.0;
	ELSIF PG.Act.PV._5.PV_Input.ManualValue_Percent < 0.0 THEN
		PG.Act.PV._5.PV_Input.ManualValue_Percent := 0.0;
	END_IF;
	IF PG.Act.PV._5.PV_Input.SP_Percent > 100.0 THEN
		PG.Act.PV._5.PV_Input.SP_Percent := 100.0;
	ELSIF PG.Act.PV._5.PV_Input.SP_Percent < 0.0 THEN
		PG.Act.PV._5.PV_Input.SP_Percent := 0.0;
	END_IF;
END_ACTION
```

#### PumpCtrl.st
```iecst
ACTION PumpCtrl:
	(* ======================================================================== *)
	(* PUMPCTRL - MANUELNA SERVISNA KOREKCIJA FREKVENCIJE                    *)
	(* MANUAL: tasteri menjaju frekvencu samo kada automatski vlasnik ne radi. *)
	(* AUTO: BRB2_rad/RB1_work zadrzavaju vlasnistvo nad regulacijom i rampom. *)
	(* COMMON: svi zahtevi se ogranicavaju na FR_min..FR_max pogona.           *)
	(* STOP/FAULT: ovaj action ne zaobilazi fault ili sigurnosno zaustavljanje. *)
	(* ======================================================================== *)
	(* ======================================================================== *)
	(* 1) Rucna korekcija frekvencije pumpi                                     *)
	(* ======================================================================== *)
	IF NOT PGRad_Cmd.Aktivan THEN
		IF EDGEPOS(Pu1_1_plus) THEN
			PG.Act.Pu._1.FR_set := PG.Act.Pu._1.FR_set + 1.0;
		END_IF;
		IF EDGEPOS(Pu1_01_plus) THEN
			PG.Act.Pu._1.FR_set := PG.Act.Pu._1.FR_set + 0.1;
		END_IF;
		IF EDGEPOS(Pu1_1_minus) THEN
			PG.Act.Pu._1.FR_set := PG.Act.Pu._1.FR_set - 1.0;
		END_IF;
		IF EDGEPOS(Pu1_01_minus) THEN
			PG.Act.Pu._1.FR_set := PG.Act.Pu._1.FR_set - 0.1;
		END_IF;

		IF EDGEPOS(Pu2_1_plus) THEN
			PG.Act.Pu._2.FR_set := PG.Act.Pu._2.FR_set + 1.0;
		END_IF;
		IF EDGEPOS(Pu2_01_plus) THEN
			PG.Act.Pu._2.FR_set := PG.Act.Pu._2.FR_set + 0.1;
		END_IF;
		IF EDGEPOS(Pu2_1_minus) THEN
			PG.Act.Pu._2.FR_set := PG.Act.Pu._2.FR_set - 1.0;
		END_IF;
		IF EDGEPOS(Pu2_01_minus) THEN
			PG.Act.Pu._2.FR_set := PG.Act.Pu._2.FR_set - 0.1;
		END_IF;
	END_IF;

	(* ======================================================================== *)
	(* 2) Granice frekvencije pumpi                                             *)
	(* ======================================================================== *)
	IF PG.Act.Pu._1.FR_set > PG.Act.Pu._1.FR_max THEN
		PG.Act.Pu._1.FR_set := PG.Act.Pu._1.FR_max;
	ELSIF PG.Act.Pu._1.FR_set < PG.Act.Pu._1.FR_min THEN
		PG.Act.Pu._1.FR_set := PG.Act.Pu._1.FR_min;
	END_IF;
	IF PG.Act.Pu._2.FR_set > PG.Act.Pu._2.FR_max THEN
		PG.Act.Pu._2.FR_set := PG.Act.Pu._2.FR_max;
	ELSIF PG.Act.Pu._2.FR_set < PG.Act.Pu._2.FR_min THEN
		PG.Act.Pu._2.FR_set := PG.Act.Pu._2.FR_min;
	END_IF;
END_ACTION
```

#### ProcessValues.st
```iecst
ACTION ProcessValues:
	(* ======================================================================== *)
	(* PROCESSVALUES - IZVEDENE PROCESNE VELICINE                            *)
	(* COMMON: racuna nivo, protok i toplotne velicine; ne komanduje opremom. *)
	(* STATUS: rezultatima se koriste Rad_PG_KB, HMI i komunikacioni ugovori.  *)
	(* ======================================================================== *)
	(* ======================================================================== *)
	(* 1) Izbor realnog protoka aktivnog izvora                                 *)
	(* ======================================================================== *)
	CASE PGRad.Ctrl.SelektovaniIzvor OF
		_01_BRB2:
			AktivniUlazniProtok := PG01_Remote.BRB2Sens.FtRB21.Value;

		_02_IEBKB1:
			AktivniUlazniProtok := IEB_KB1.Cntrl.Comm.Podstanica.Status.TrenutniProtok;

	ELSE
		AktivniUlazniProtok := 0.0;
	END_CASE

	(* ======================================================================== *)
	(* 2) Toplotne snage                                                        *)
	(* ======================================================================== *)
	(* 4.181 je specificni toplotni kapacitet vode; uz protok [l/s] i delta T [degC] rezultat je [kW]. *)
	Predata_Snaga := 4.181 * (*AktivniUlazniProtok*) PG.Sens.MP._1.AI_Output.ScaledValue
		* (PG.Sens.Tt._1.AI_Output.ScaledValue - PG.Sens.Tt._2.AI_Output.ScaledValue);
	Snaga_grejanja_hotela := 4.181 * (*AktivniUlazniProtok*) PG.Sens.MP._1.AI_Output.ScaledValue
		* (PG.Sens.Tt._1.AI_Output.ScaledValue - PG.Sens.Tt._4.AI_Output.ScaledValue);
	Snaga_sanitarnog_grejanja := Predata_Snaga - Snaga_grejanja_hotela;

	(* ======================================================================== *)
	(* 3) Ostale izvedene procesne velicine                                     *)
	(* ======================================================================== *)
	(* Faktor 0.09804 pretvara diferencijalni hidrostatski pritisak [bar] u nivo vode [m]. *)
	NivoPrihvatniSud := (PG.Sens.Pt._NS1.AI_Output.ScaledValue - PG.Sens.Pt._NS2.AI_Output.ScaledValue) / 0.09804;
	(* 0.123 je postojeca commissioning korekcija DP strainer-a; fizicko poreklo treba potvrditi. *)
	DP_strainer := PG.Sens.Pt._1.AI_Output.ScaledValue - PG.Sens.Pt._2.AI_Output.ScaledValue + 0.123;
	(* 0.0015 je postojeca commissioning korekcija DP izmenjivaca; fizicko poreklo treba potvrditi. *)
	DP_Izmejnivac := PG.Sens.Pt._2.AI_Output.ScaledValue - PG.Sens.Pt._3.AI_Output.ScaledValue + 0.0015;
END_ACTION
```

### Program Logical/Project/Rad_PG_KB (IEC)
